LIN {X 0,Y 291.347,Z 435.191,A -85,B 0,C 180,E1 -16863.698,E2 -16863.698} C_VEL
LIN {X 0,Y 291.408,Z 435.188,A -85,B 0,C 180,E1 -16867.262,E2 -16867.262} C_VEL
LIN {X 0,Y 291.407,Z 435.186,A -85,B 0,C 180,E1 -16870.63,E2 -16870.63} C_VEL
LIN {X 0,Y 291.354,Z 435.191,A -85,B 0,C 180,E1 -16874.39,E2 -16874.39} C_VEL
LIN {X 0,Y 291.333,Z 435.194,A -85,B 0,C 180,E1 -16878.403,E2 -16878.403} C_VEL
LIN {X 0,Y 291.349,Z 435.194,A -85,B 0,C 180,E1 -16881.157,E2 -16881.157} C_VEL
LIN {X 0,Y 291.362,Z 435.192,A -85,B 0,C 180,E1 -16884.626,E2 -16884.626} C_VEL
LIN {X 0,Y 291.372,Z 435.186,A -85,B 0,C 180,E1 -16887.951,E2 -16887.951} C_VEL
LIN {X 0,Y 291.379,Z 435.188,A -85,B 0,C 180,E1 -16891.158,E2 -16891.158} C_VEL
LIN {X 0,Y 291.414,Z 435.184,A -85,B 0,C 180,E1 -16894.272,E2 -16894.272} C_VEL
LIN {X 0,Y 291.384,Z 435.184,A -85,B 0,C 180,E1 -16897.3,E2 -16897.3} C_VEL
LIN {X 0,Y 291.46,Z 435.179,A -85,B 0,C 180,E1 -16900.27,E2 -16900.27} C_VEL
LIN {X 0,Y 291.557,Z 435.169,A -85,B 0,C 180,E1 -16904.624,E2 -16904.624} C_VEL
LIN {X 0,Y 291.539,Z 435.169,A -85,B 0,C 180,E1 -16908.881,E2 -16908.881} C_VEL
LIN {X 0,Y 291.67,Z 435.151,A -85,B 0,C 180,E1 -16911.687,E2 -16911.687} C_VEL
LIN {X 0,Y 291.627,Z 435.154,A -85,B 0,C 180,E1 -16914.468,E2 -16914.468} C_VEL
LIN {X 0,Y 291.892,Z 435.126,A -85,B 0,C 180,E1 -16918.62,E2 -16918.62} C_VEL
LIN {X 0,Y 291.893,Z 435.118,A -85,B 0,C 180,E1 -16921.38,E2 -16921.38} C_VEL
LIN {X 0,Y 291.556,Z 435.166,A -85,B 0,C 180,E1 -16924.218,E2 -16924.218} C_VEL
LIN {X 0,Y 290.899,Z 435.248,A -85,B 0,C 180,E1 -16925.372,E2 -16925.372} C_VEL
LIN {X 0,Y 288.07,Z 435.598,A -85,B 0,C 180,E1 -16927.252,E2 -16927.252} C_VEL
LIN {X 0,Y 285.651,Z 435.902,A -85,B 0,C 180,E1 -16928.777,E2 -16928.777} C_VEL
LIN {X 0,Y 284.591,Z 436.034,A -85,B 0,C 180,E1 -16929.959,E2 -16929.959} C_VEL
LIN {X 0,Y 284.493,Z 436.044,A -85,B 0,C 180,E1 -16930.36,E2 -16930.36} C_VEL
LIN {X 0,Y 284.484,Z 436.05,A -85,B 0,C 180,E1 -16934.303,E2 -16934.303} C_VEL
LIN {X 0,Y 284.427,Z 436.051,A -85,B 0,C 180,E1 -16937.248,E2 -16937.248} C_VEL
LIN {X 0,Y 284.379,Z 436.064,A -85,B 0,C 180,E1 -16940.242,E2 -16940.242} C_VEL
LIN {X 0,Y 284.34,Z 436.065,A -85,B 0,C 180,E1 -16944.846,E2 -16944.846} C_VEL
LIN {X 0,Y 284.331,Z 436.069,A -85,B 0,C 180,E1 -16948.011,E2 -16948.011} C_VEL
LIN {X 0,Y 284.295,Z 436.072,A -85,B 0,C 180,E1 -16951.274,E2 -16951.274} C_VEL
LIN {X 0,Y 284.363,Z 436.065,A -85,B 0,C 180,E1 -16955.354,E2 -16955.354} C_VEL
LIN {X 0,Y 284.368,Z 436.211,A -85,B 0,C 180,E1 -16958.839,E2 -16958.839} C_VEL
LIN {X 0,Y 285.634,Z 442.53,A -85,B 0,C 180,E1 -16962.426,E2 -16962.426} C_VEL
LIN {X 0,Y 287.31,Z 450.763,A -85,B 0,C 180,E1 -16966.771,E2 -16966.771} C_VEL
LIN {X 0,Y 288.547,Z 457.203,A -85,B 0,C 180,E1 -16969.939,E2 -16969.939} C_VEL
LIN {X 0,Y 288.86,Z 459.714,A -85,B 0,C 180,E1 -16971.13,E2 -16971.13} C_VEL
LIN {X 0,Y 288.1,Z 465.339,A -85,B 0,C 180,E1 -16973.612,E2 -16973.612} C_VEL
LIN {X 0,Y 286.625,Z 474.02,A -85,B 0,C 180,E1 -16977.355,E2 -16977.355} C_VEL
LIN {X 0,Y 285.082,Z 485.04,A -85,B 0,C 180,E1 -16982.07,E2 -16982.07} C_VEL
LIN {X 0,Y 284.576,Z 489.714,A -85,B 0,C 180,E1 -16984.074,E2 -16984.074} C_VEL
LIN {X 0,Y 287.073,Z 505.085,A -85,B 0,C 180,E1 -16984.981,E2 -16984.981} C_VEL
LIN {X 0,Y 288.406,Z 518.048,A -85,B 0,C 180,E1 -16985.981,E2 -16985.981} C_VEL
LIN {X 0,Y 288.965,Z 530.807,A -85,B 0,C 180,E1 -16987.206,E2 -16987.206} C_VEL
LIN {X 0,Y 288.929,Z 542.594,A -85,B 0,C 180,E1 -16988.601,E2 -16988.601} C_VEL
LIN {X 0,Y 288.46,Z 553.824,A -85,B 0,C 180,E1 -16990.242,E2 -16990.242} C_VEL
LIN {X 0,Y 287.04,Z 562.869,A -85,B 0,C 180,E1 -16991.81,E2 -16991.81} C_VEL
LIN {X 0,Y 285.561,Z 571.816,A -85,B 0,C 180,E1 -16993.707,E2 -16993.707} C_VEL
LIN {X 0,Y 284.788,Z 576.889,A -85,B 0,C 180,E1 -16994.982,E2 -16994.982} C_VEL
LIN {X 0,Y 283.886,Z 583.999,A -85,B 0,C 180,E1 -16997.126,E2 -16997.126} C_VEL
LIN {X 0,Y 283.299,Z 589.729,A -85,B 0,C 180,E1 -16999.277,E2 -16999.277} C_VEL
LIN {X 0,Y 283.176,Z 594.281,A -85,B 0,C 180,E1 -17001.436,E2 -17001.436} C_VEL
LIN {X 0,Y 283.275,Z 596.802,A -85,B 0,C 180,E1 -17002.93,E2 -17002.93} C_VEL
LIN {X 0,Y 283.396,Z 598.695,A -85,B 0,C 180,E1 -17004.307,E2 -17004.307} C_VEL
LIN {X 0,Y 283.685,Z 600.209,A -85,B 0,C 180,E1 -17005.738,E2 -17005.738} C_VEL
LIN {X 0,Y 283.839,Z 601.281,A -85,B 0,C 180,E1 -17007.162,E2 -17007.162} C_VEL
LIN {X 0,Y 284.353,Z 602.219,A -85,B 0,C 180,E1 -17010,E2 -17010} C_VEL
LIN {X 0,Y 283.84,Z 601.271,A -85,B 0,C 180,E1 -17012.839,E2 -17012.839} C_VEL
LIN {X 0,Y 283.684,Z 600.194,A -85,B 0,C 180,E1 -17014.262,E2 -17014.262} C_VEL
LIN {X 0,Y 283.39,Z 598.672,A -85,B 0,C 180,E1 -17015.693,E2 -17015.693} C_VEL
LIN {X 0,Y 283.199,Z 595.541,A -85,B 0,C 180,E1 -17017.845,E2 -17017.845} C_VEL
LIN {X 0,Y 283.227,Z 591.348,A -85,B 0,C 180,E1 -17020.003,E2 -17020.003} C_VEL
LIN {X 0,Y 283.741,Z 584.975,A -85,B 0,C 180,E1 -17022.517,E2 -17022.517} C_VEL
LIN {X 0,Y 284.62,Z 578.08,A -85,B 0,C 180,E1 -17024.661,E2 -17024.661} C_VEL
LIN {X 0,Y 285.383,Z 572.557,A -85,B 0,C 180,E1 -17026.099,E2 -17026.099} C_VEL
LIN {X 0,Y 286.766,Z 564.569,A -85,B 0,C 180,E1 -17027.839,E2 -17027.839} C_VEL
LIN {X 0,Y 288.329,Z 554.77,A -85,B 0,C 180,E1 -17029.582,E2 -17029.582} C_VEL
LIN {X 0,Y 288.853,Z 543.762,A -85,B 0,C 180,E1 -17031.218,E2 -17031.218} C_VEL
LIN {X 0,Y 289.008,Z 533.538,A -85,B 0,C 180,E1 -17032.471,E2 -17032.471} C_VEL
LIN {X 0,Y 288.596,Z 521.211,A -85,B 0,C 180,E1 -17033.716,E2 -17033.716} C_VEL
LIN {X 0,Y 287.262,Z 507.25,A -85,B 0,C 180,E1 -17034.842,E2 -17034.842} C_VEL
LIN {X 0,Y 285.279,Z 494.142,A -85,B 0,C 180,E1 -17035.667,E2 -17035.667} C_VEL
LIN {X 0,Y 284.558,Z 489.7,A -85,B 0,C 180,E1 -17035.902,E2 -17035.902} C_VEL
LIN {X 0,Y 286.053,Z 477.671,A -85,B 0,C 180,E1 -17041.061,E2 -17041.061} C_VEL
LIN {X 0,Y 287.257,Z 470.208,A -85,B 0,C 180,E1 -17044.244,E2 -17044.244} C_VEL
LIN {X 0,Y 288.78,Z 461.165,A -85,B 0,C 180,E1 -17048.176,E2 -17048.176} C_VEL
LIN {X 0,Y 288.817,Z 458.788,A -85,B 0,C 180,E1 -17049.248,E2 -17049.248} C_VEL
LIN {X 0,Y 287.42,Z 451.508,A -85,B 0,C 180,E1 -17052.814,E2 -17052.814} C_VEL
LIN {X 0,Y 285.966,Z 444.403,A -85,B 0,C 180,E1 -17056.517,E2 -17056.517} C_VEL
LIN {X 0,Y 284.724,Z 437.997,A -85,B 0,C 180,E1 -17060.076,E2 -17060.076} C_VEL
LIN {X 0,Y 284.329,Z 436.071,A -85,B 0,C 180,E1 -17061.269,E2 -17061.269} C_VEL
LIN {X 0,Y 284.364,Z 436.063,A -85,B 0,C 180,E1 -17064.646,E2 -17064.646} C_VEL
LIN {X 0,Y 284.297,Z 436.069,A -85,B 0,C 180,E1 -17068.726,E2 -17068.726} C_VEL
LIN {X 0,Y 284.399,Z 436.06,A -85,B 0,C 180,E1 -17072.827,E2 -17072.827} C_VEL
LIN {X 0,Y 284.336,Z 436.065,A -85,B 0,C 180,E1 -17076.704,E2 -17076.704} C_VEL
LIN {X 0,Y 284.406,Z 436.057,A -85,B 0,C 180,E1 -17081.262,E2 -17081.262} C_VEL
LIN {X 0,Y 284.495,Z 436.047,A -85,B 0,C 180,E1 -17084.459,E2 -17084.459} C_VEL
LIN {X 0,Y 284.492,Z 436.047,A -85,B 0,C 180,E1 -17088.602,E2 -17088.602} C_VEL
LIN {X 0,Y 284.625,Z 436.032,A -85,B 0,C 180,E1 -17091.48,E2 -17091.48} C_VEL
LIN {X 0,Y 284.598,Z 436.034,A -85,B 0,C 180,E1 -17094.331,E2 -17094.331} C_VEL
LIN {X 0,Y 284.86,Z 436,A -85,B 0,C 180,E1 -17098.586,E2 -17098.586} C_VEL
LIN {X 0,Y 284.859,Z 436.002,A -85,B 0,C 180,E1 -17101.414,E2 -17101.414} C_VEL
LIN {X 0,Y 284.677,Z 436.023,A -85,B 0,C 180,E1 -17107.091,E2 -17107.091} C_VEL
LIN {X 0,Y 284.521,Z 436.042,A -85,B 0,C 180,E1 -17109.957,E2 -17109.957} C_VEL
LIN {X 0,Y 284.486,Z 436.028,A -85,B 0,C 180,E1 -17114.303,E2 -17114.303} C_VEL
LIN {X 0,Y 284.428,Z 436.036,A -85,B 0,C 180,E1 -17117.248,E2 -17117.248} C_VEL
LIN {X 0,Y 284.382,Z 436.056,A -85,B 0,C 180,E1 -17120.242,E2 -17120.242} C_VEL
LIN {X 0,Y 284.372,Z 436.056,A -85,B 0,C 180,E1 -17123.875,E2 -17123.875} C_VEL
LIN {X 0,Y 284.397,Z 436.041,A -85,B 0,C 180,E1 -17127.172,E2 -17127.172} C_VEL
LIN {X 0,Y 284.296,Z 436.069,A -85,B 0,C 180,E1 -17131.274,E2 -17131.274} C_VEL
LIN {X 0,Y 284.343,Z 436.064,A -85,B 0,C 180,E1 -17135.348,E2 -17135.348} C_VEL
LIN {X 0,Y 284.311,Z 436.068,A -85,B 0,C 180,E1 -17138.169,E2 -17138.169} C_VEL
LIN {X 0,Y 284.286,Z 436.071,A -85,B 0,C 180,E1 -17142.128,E2 -17142.128} C_VEL
LIN {X 0,Y 284.32,Z 436.066,A -85,B 0,C 180,E1 -17146.201,E2 -17146.201} C_VEL
LIN {X 0,Y 284.354,Z 436.06,A -85,B 0,C 180,E1 -17150.013,E2 -17150.013} C_VEL
LIN {X 0,Y 284.358,Z 436.059,A -85,B 0,C 180,E1 -17153.618,E2 -17153.618} C_VEL
LIN {X 0,Y 284.31,Z 436.069,A -85,B 0,C 180,E1 -17157.19,E2 -17157.19} C_VEL
LIN {X 0,Y 284.358,Z 436.063,A -85,B 0,C 180,E1 -17160.376,E2 -17160.376} C_VEL
LIN {X 0,Y 284.389,Z 436.062,A -85,B 0,C 180,E1 -17164.375,E2 -17164.375} C_VEL
LIN {X 0,Y 284.416,Z 436.147,A -85,B 0,C 180,E1 -17165.136,E2 -17165.136} C_VEL
LIN {X 0,Y 287.692,Z 444.694,A -85,B 0,C 180,E1 -17166.157,E2 -17166.157} C_VEL
LIN {X 0,Y 291.581,Z 455.705,A -85,B 0,C 180,E1 -17167.66,E2 -17167.66} C_VEL
LIN {X 0,Y 294.434,Z 465.794,A -85,B 0,C 180,E1 -17169.236,E2 -17169.236} C_VEL
LIN {X 0,Y 294.248,Z 468.913,A -85,B 0,C 180,E1 -17169.676,E2 -17169.676} C_VEL
LIN {X 0,Y 292.847,Z 478.165,A -85,B 0,C 180,E1 -17171.096,E2 -17171.096} C_VEL
LIN {X 0,Y 291.409,Z 487.197,A -85,B 0,C 180,E1 -17172.816,E2 -17172.816} C_VEL
LIN {X 0,Y 289.663,Z 495.979,A -85,B 0,C 180,E1 -17174.881,E2 -17174.881} C_VEL
LIN {X 0,Y 288.283,Z 503.021,A -85,B 0,C 180,E1 -17176.967,E2 -17176.967} C_VEL
LIN {X 0,Y 287.359,Z 507.755,A -85,B 0,C 180,E1 -17178.717,E2 -17178.717} C_VEL
LIN {X 0,Y 286.426,Z 512.352,A -85,B 0,C 180,E1 -17180.823,E2 -17180.823} C_VEL
LIN {X 0,Y 285.582,Z 515.883,A -85,B 0,C 180,E1 -17182.932,E2 -17182.932} C_VEL
LIN {X 0,Y 285.161,Z 517.704,A -85,B 0,C 180,E1 -17184.342,E2 -17184.342} C_VEL
LIN {X 0,Y 284.821,Z 519.076,A -85,B 0,C 180,E1 -17185.755,E2 -17185.755} C_VEL
LIN {X 0,Y 284.762,Z 520.603,A -85,B 0,C 180,E1 -17188.586,E2 -17188.586} C_VEL
LIN {X 0,Y 284.742,Z 520.826,A -85,B 0,C 180,E1 -17190,E2 -17190} C_VEL
LIN {X 0,Y 284.761,Z 520.64,A -85,B 0,C 180,E1 -17191.414,E2 -17191.414} C_VEL
LIN {X 0,Y 284.812,Z 519.162,A -85,B 0,C 180,E1 -17194.245,E2 -17194.245} C_VEL
LIN {X 0,Y 285.147,Z 517.83,A -85,B 0,C 180,E1 -17195.658,E2 -17195.658} C_VEL
LIN {X 0,Y 285.867,Z 515.009,A -85,B 0,C 180,E1 -17197.771,E2 -17197.771} C_VEL
LIN {X 0,Y 286.759,Z 511.19,A -85,B 0,C 180,E1 -17199.878,E2 -17199.878} C_VEL
LIN {X 0,Y 287.795,Z 505.275,A -85,B 0,C 180,E1 -17202.363,E2 -17202.363} C_VEL
LIN {X 0,Y 289.175,Z 498.879,A -85,B 0,C 180,E1 -17204.425,E2 -17204.425} C_VEL
LIN {X 0,Y 290.779,Z 490.841,A -85,B 0,C 180,E1 -17206.499,E2 -17206.499} C_VEL
LIN {X 0,Y 292.119,Z 482.62,A -85,B 0,C 180,E1 -17208.226,E2 -17208.226} C_VEL
LIN {X 0,Y 293.692,Z 472.862,A -85,B 0,C 180,E1 -17209.867,E2 -17209.867} C_VEL
LIN {X 0,Y 294.51,Z 466.371,A -85,B 0,C 180,E1 -17210.791,E2 -17210.791} C_VEL
LIN {X 0,Y 291.709,Z 456.12,A -85,B 0,C 180,E1 -17212.399,E2 -17212.399} C_VEL
LIN {X 0,Y 288.801,Z 447.537,A -85,B 0,C 180,E1 -17213.592,E2 -17213.592} C_VEL
LIN {X 0,Y 284.726,Z 437.456,A -85,B 0,C 180,E1 -17214.859,E2 -17214.859} C_VEL
LIN {X 0,Y 284.419,Z 436.058,A -85,B 0,C 180,E1 -17215.034,E2 -17215.034} C_VEL
LIN {X 0,Y 284.33,Z 436.06,A -85,B 0,C 180,E1 -17218.011,E2 -17218.011} C_VEL
LIN {X 0,Y 284.296,Z 436.07,A -85,B 0,C 180,E1 -17221.274,E2 -17221.274} C_VEL
LIN {X 0,Y 284.364,Z 436.063,A -85,B 0,C 180,E1 -17225.354,E2 -17225.354} C_VEL
LIN {X 0,Y 284.341,Z 436.065,A -85,B 0,C 180,E1 -17228.165,E2 -17228.165} C_VEL
LIN {X 0,Y 284.344,Z 436.064,A -85,B 0,C 180,E1 -17232.141,E2 -17232.141} C_VEL
LIN {X 0,Y 284.298,Z 436.07,A -85,B 0,C 180,E1 -17236.197,E2 -17236.197} C_VEL
LIN {X 0,Y 284.308,Z 436.068,A -85,B 0,C 180,E1 -17240.024,E2 -17240.024} C_VEL
LIN {X 0,Y 284.332,Z 436.065,A -85,B 0,C 180,E1 -17243.614,E2 -17243.614} C_VEL
LIN {X 0,Y 284.309,Z 436.067,A -85,B 0,C 180,E1 -17247.19,E2 -17247.19} C_VEL
LIN {X 0,Y 284.357,Z 436.064,A -85,B 0,C 180,E1 -17250.376,E2 -17250.376} C_VEL
LIN {X 0,Y 284.376,Z 436.059,A -85,B 0,C 180,E1 -17253.586,E2 -17253.586} C_VEL
LIN {X 0,Y 284.368,Z 436.062,A -85,B 0,C 180,E1 -17256.707,E2 -17256.707} C_VEL
LIN {X 0,Y 284.406,Z 436.055,A -85,B 0,C 180,E1 -17261.262,E2 -17261.262} C_VEL
LIN {X 0,Y 284.494,Z 436.047,A -85,B 0,C 180,E1 -17264.459,E2 -17264.459} C_VEL
LIN {X 0,Y 284.491,Z 436.046,A -85,B 0,C 180,E1 -17268.601,E2 -17268.601} C_VEL
LIN {X 0,Y 284.624,Z 436.029,A -85,B 0,C 180,E1 -17271.48,E2 -17271.48} C_VEL
LIN {X 0,Y 284.597,Z 436.029,A -85,B 0,C 180,E1 -17274.331,E2 -17274.331} C_VEL
LIN {X 0,Y 284.858,Z 436.003,A -85,B 0,C 180,E1 -17278.586,E2 -17278.586} C_VEL
LIN {X 0,Y 284.859,Z 435.994,A -85,B 0,C 180,E1 -17281.414,E2 -17281.414} C_VEL
LIN {X 0,Y 284.676,Z 436.019,A -85,B 0,C 180,E1 -17287.091,E2 -17287.091} C_VEL
LIN {X 0,Y 284.493,Z 436.044,A -85,B 0,C 180,E1 -17290.36,E2 -17290.36} C_VEL
LIN {X 0,Y 283.799,Z 436.132,A -85,B 0,C 180,E1 -17291.541,E2 -17291.541} C_VEL
LIN {X 0,Y 280.951,Z 436.486,A -85,B 0,C 180,E1 -17293.466,E2 -17293.466} C_VEL
LIN {X 0,Y 278.535,Z 436.789,A -85,B 0,C 180,E1 -17295.029,E2 -17295.029} C_VEL
LIN {X 0,Y 277.474,Z 436.921,A -85,B 0,C 180,E1 -17296.239,E2 -17296.239} C_VEL
LIN {X 0,Y 277.373,Z 436.93,A -85,B 0,C 180,E1 -17296.65,E2 -17296.65} C_VEL
LIN {X 0,Y 277.292,Z 436.944,A -85,B 0,C 180,E1 -17300.783,E2 -17300.783} C_VEL
LIN {X 0,Y 277.294,Z 436.947,A -85,B 0,C 180,E1 -17304.158,E2 -17304.158} C_VEL
LIN {X 0,Y 277.326,Z 436.94,A -85,B 0,C 180,E1 -17307.505,E2 -17307.505} C_VEL
LIN {X 0,Y 277.273,Z 436.948,A -85,B 0,C 180,E1 -17310.481,E2 -17310.481} C_VEL
LIN {X 0,Y 277.255,Z 436.95,A -85,B 0,C 180,E1 -17313.895,E2 -17313.895} C_VEL
LIN {X 0,Y 277.283,Z 436.946,A -85,B 0,C 180,E1 -17317.467,E2 -17317.467} C_VEL
LIN {X 0,Y 277.322,Z 437.139,A -85,B 0,C 180,E1 -17318.222,E2 -17318.222} C_VEL
LIN {X 0,Y 278.6,Z 443.48,A -85,B 0,C 180,E1 -17321.951,E2 -17321.951} C_VEL
LIN {X 0,Y 280.048,Z 450.645,A -85,B 0,C 180,E1 -17325.874,E2 -17325.874} C_VEL
LIN {X 0,Y 281.663,Z 459.053,A -85,B 0,C 180,E1 -17330.156,E2 -17330.156} C_VEL
LIN {X 0,Y 281.813,Z 461.726,A -85,B 0,C 180,E1 -17331.43,E2 -17331.43} C_VEL
LIN {X 0,Y 280.511,Z 469.265,A -85,B 0,C 180,E1 -17334.813,E2 -17334.813} C_VEL
LIN {X 0,Y 278.965,Z 478.58,A -85,B 0,C 180,E1 -17338.933,E2 -17338.933} C_VEL
LIN {X 0,Y 277.645,Z 488.643,A -85,B 0,C 180,E1 -17343.379,E2 -17343.379} C_VEL
LIN {X 0,Y 280.156,Z 503.724,A -85,B 0,C 180,E1 -17344.303,E2 -17344.303} C_VEL
LIN {X 0,Y 281.504,Z 516.559,A -85,B 0,C 180,E1 -17345.318,E2 -17345.318} C_VEL
LIN {X 0,Y 282.114,Z 528.716,A -85,B 0,C 180,E1 -17346.51,E2 -17346.51} C_VEL
LIN {X 0,Y 282.129,Z 540.026,A -85,B 0,C 180,E1 -17347.859,E2 -17347.859} C_VEL
LIN {X 0,Y 281.677,Z 550.499,A -85,B 0,C 180,E1 -17349.364,E2 -17349.364} C_VEL
LIN {X 0,Y 281.112,Z 557.048,A -85,B 0,C 180,E1 -17350.465,E2 -17350.465} C_VEL
LIN {X 0,Y 279.385,Z 567.046,A -85,B 0,C 180,E1 -17352.43,E2 -17352.43} C_VEL
LIN {X 0,Y 277.789,Z 575.855,A -85,B 0,C 180,E1 -17354.595,E2 -17354.595} C_VEL
LIN {X 0,Y 276.862,Z 582.969,A -85,B 0,C 180,E1 -17356.794,E2 -17356.794} C_VEL
LIN {X 0,Y 276.249,Z 588.704,A -85,B 0,C 180,E1 -17359,E2 -17359} C_VEL
LIN {X 0,Y 276.115,Z 593.26,A -85,B 0,C 180,E1 -17361.216,E2 -17361.216} C_VEL
LIN {X 0,Y 276.204,Z 596.035,A -85,B 0,C 180,E1 -17362.912,E2 -17362.912} C_VEL
LIN {X 0,Y 276.599,Z 599.193,A -85,B 0,C 180,E1 -17365.628,E2 -17365.628} C_VEL
LIN {X 0,Y 276.783,Z 600.271,A -85,B 0,C 180,E1 -17367.089,E2 -17367.089} C_VEL
LIN {X 0,Y 277.321,Z 601.213,A -85,B 0,C 180,E1 -17370,E2 -17370} C_VEL
LIN {X 0,Y 276.783,Z 600.26,A -85,B 0,C 180,E1 -17372.911,E2 -17372.911} C_VEL
LIN {X 0,Y 276.597,Z 599.177,A -85,B 0,C 180,E1 -17374.372,E2 -17374.372} C_VEL
LIN {X 0,Y 276.208,Z 595.994,A -85,B 0,C 180,E1 -17377.095,E2 -17377.095} C_VEL
LIN {X 0,Y 276.121,Z 591.827,A -85,B 0,C 180,E1 -17379.523,E2 -17379.523} C_VEL
LIN {X 0,Y 276.403,Z 586.875,A -85,B 0,C 180,E1 -17381.737,E2 -17381.737} C_VEL
LIN {X 0,Y 277.27,Z 579.519,A -85,B 0,C 180,E1 -17384.308,E2 -17384.308} C_VEL
LIN {X 0,Y 278.203,Z 573.005,A -85,B 0,C 180,E1 -17386.134,E2 -17386.134} C_VEL
LIN {X 0,Y 279.649,Z 565.264,A -85,B 0,C 180,E1 -17387.931,E2 -17387.931} C_VEL
LIN {X 0,Y 281.203,Z 555.896,A -85,B 0,C 180,E1 -17389.719,E2 -17389.719} C_VEL
LIN {X 0,Y 281.922,Z 545.374,A -85,B 0,C 180,E1 -17391.382,E2 -17391.382} C_VEL
LIN {X 0,Y 282.183,Z 534.115,A -85,B 0,C 180,E1 -17392.851,E2 -17392.851} C_VEL
LIN {X 0,Y 281.879,Z 522.439,A -85,B 0,C 180,E1 -17394.107,E2 -17394.107} C_VEL
LIN {X 0,Y 280.911,Z 510.397,A -85,B 0,C 180,E1 -17395.171,E2 -17395.171} C_VEL
LIN {X 0,Y 279.154,Z 497.2,A -85,B 0,C 180,E1 -17396.097,E2 -17396.097} C_VEL
LIN {X 0,Y 277.639,Z 488.645,A -85,B 0,C 180,E1 -17396.583,E2 -17396.583} C_VEL
LIN {X 0,Y 278.951,Z 478.521,A -85,B 0,C 180,E1 -17401.062,E2 -17401.062} C_VEL
LIN {X 0,Y 280.494,Z 469.171,A -85,B 0,C 180,E1 -17405.19,E2 -17405.19} C_VEL
LIN {X 0,Y 281.814,Z 461.628,A -85,B 0,C 180,E1 -17408.57,E2 -17408.57} C_VEL
LIN {X 0,Y 281.66,Z 458.923,A -85,B 0,C 180,E1 -17409.844,E2 -17409.844} C_VEL
LIN {X 0,Y 280.328,Z 452.037,A -85,B 0,C 180,E1 -17413.36,E2 -17413.36} C_VEL
LIN {X 0,Y 278.862,Z 445.062,A -85,B 0,C 180,E1 -17417.12,E2 -17417.12} C_VEL
LIN {X 0,Y 277.662,Z 438.766,A -85,B 0,C 180,E1 -17420.744,E2 -17420.744} C_VEL
LIN {X 0,Y 277.291,Z 436.949,A -85,B 0,C 180,E1 -17421.91,E2 -17421.91} C_VEL
LIN {X 0,Y 277.306,Z 436.943,A -85,B 0,C 180,E1 -17424.345,E2 -17424.345} C_VEL
LIN {X 0,Y 277.246,Z 436.952,A -85,B 0,C 180,E1 -17427.837,E2 -17427.837} C_VEL
LIN {X 0,Y 277.271,Z 436.948,A -85,B 0,C 180,E1 -17431.21,E2 -17431.21} C_VEL
LIN {X 0,Y 277.312,Z 436.94,A -85,B 0,C 180,E1 -17434.479,E2 -17434.479} C_VEL
LIN {X 0,Y 277.271,Z 436.946,A -85,B 0,C 180,E1 -17437.654,E2 -17437.654} C_VEL
LIN {X 0,Y 277.347,Z 436.935,A -85,B 0,C 180,E1 -17440.766,E2 -17440.766} C_VEL
LIN {X 0,Y 277.438,Z 436.927,A -85,B 0,C 180,E1 -17445.326,E2 -17445.326} C_VEL
LIN {X 0,Y 277.463,Z 436.927,A -85,B 0,C 180,E1 -17449.787,E2 -17449.787} C_VEL
LIN {X 0,Y 277.632,Z 436.902,A -85,B 0,C 180,E1 -17452.729,E2 -17452.729} C_VEL
LIN {X 0,Y 277.826,Z 436.877,A -85,B 0,C 180,E1 -17458.551,E2 -17458.551} C_VEL
LIN {X 0,Y 277.825,Z 436.879,A -85,B 0,C 180,E1 -17461.45,E2 -17461.45} C_VEL
LIN {X 0,Y 277.631,Z 436.902,A -85,B 0,C 180,E1 -17467.272,E2 -17467.272} C_VEL
LIN {X 0,Y 277.464,Z 436.92,A -85,B 0,C 180,E1 -17470.213,E2 -17470.213} C_VEL
LIN {X 0,Y 277.438,Z 436.904,A -85,B 0,C 180,E1 -17474.674,E2 -17474.674} C_VEL
LIN {X 0,Y 277.348,Z 436.928,A -85,B 0,C 180,E1 -17479.234,E2 -17479.234} C_VEL
LIN {X 0,Y 277.322,Z 436.933,A -85,B 0,C 180,E1 -17484.17,E2 -17484.17} C_VEL
LIN {X 0,Y 277.325,Z 436.918,A -85,B 0,C 180,E1 -17487.504,E2 -17487.504} C_VEL
LIN {X 0,Y 277.274,Z 436.937,A -85,B 0,C 180,E1 -17490.481,E2 -17490.481} C_VEL
LIN {X 0,Y 277.249,Z 436.946,A -85,B 0,C 180,E1 -17493.896,E2 -17493.896} C_VEL
LIN {X 0,Y 277.268,Z 436.948,A -85,B 0,C 180,E1 -17497.47,E2 -17497.47} C_VEL
LIN {X 0,Y 277.218,Z 436.955,A -85,B 0,C 180,E1 -17501.235,E2 -17501.235} C_VEL
LIN {X 0,Y 277.249,Z 436.951,A -85,B 0,C 180,E1 -17505.217,E2 -17505.217} C_VEL
LIN {X 0,Y 277.297,Z 436.94,A -85,B 0,C 180,E1 -17509.494,E2 -17509.494} C_VEL
LIN {X 0,Y 277.294,Z 436.941,A -85,B 0,C 180,E1 -17512.535,E2 -17512.535} C_VEL
LIN {X 0,Y 277.257,Z 436.943,A -85,B 0,C 180,E1 -17516.105,E2 -17516.105} C_VEL
LIN {X 0,Y 277.264,Z 436.946,A -85,B 0,C 180,E1 -17519.539,E2 -17519.539} C_VEL
LIN {X 0,Y 277.346,Z 436.939,A -85,B 0,C 180,E1 -17523.675,E2 -17523.675} C_VEL
LIN {X 0,Y 277.356,Z 436.937,A -85,B 0,C 180,E1 -17524.433,E2 -17524.433} C_VEL
LIN {X 0,Y 281.583,Z 447.834,A -85,B 0,C 180,E1 -17525.806,E2 -17525.806} C_VEL
LIN {X 0,Y 285.395,Z 458.984,A -85,B 0,C 180,E1 -17527.436,E2 -17527.436} C_VEL
LIN {X 0,Y 287.67,Z 467.111,A -85,B 0,C 180,E1 -17528.766,E2 -17528.766} C_VEL
LIN {X 0,Y 287.86,Z 468.825,A -85,B 0,C 180,E1 -17529.044,E2 -17529.044} C_VEL
LIN {X 0,Y 286.208,Z 479.174,A -85,B 0,C 180,E1 -17530.64,E2 -17530.64} C_VEL
LIN {X 0,Y 284.703,Z 488.204,A -85,B 0,C 180,E1 -17532.398,E2 -17532.398} C_VEL
LIN {X 0,Y 282.885,Z 496.986,A -85,B 0,C 180,E1 -17534.51,E2 -17534.51} C_VEL
LIN {X 0,Y 281.441,Z 504.028,A -85,B 0,C 180,E1 -17536.645,E2 -17536.645} C_VEL
LIN {X 0,Y 280.47,Z 508.762,A -85,B 0,C 180,E1 -17538.436,E2 -17538.436} C_VEL
LIN {X 0,Y 279.491,Z 513.358,A -85,B 0,C 180,E1 -17540.593,E2 -17540.593} C_VEL
LIN {X 0,Y 278.609,Z 516.889,A -85,B 0,C 180,E1 -17542.754,E2 -17542.754} C_VEL
LIN {X 0,Y 278.168,Z 518.71,A -85,B 0,C 180,E1 -17544.2,E2 -17544.2} C_VEL
LIN {X 0,Y 277.813,Z 520.081,A -85,B 0,C 180,E1 -17545.647,E2 -17545.647} C_VEL
LIN {X 0,Y 277.739,Z 521.608,A -85,B 0,C 180,E1 -17548.55,E2 -17548.55} C_VEL
LIN {X 0,Y 277.717,Z 521.83,A -85,B 0,C 180,E1 -17550,E2 -17550} C_VEL
LIN {X 0,Y 277.738,Z 521.645,A -85,B 0,C 180,E1 -17551.45,E2 -17551.45} C_VEL
LIN {X 0,Y 277.804,Z 520.167,A -85,B 0,C 180,E1 -17554.353,E2 -17554.353} C_VEL
LIN {X 0,Y 278.153,Z 518.834,A -85,B 0,C 180,E1 -17555.8,E2 -17555.8} C_VEL
LIN {X 0,Y 278.906,Z 516.013,A -85,B 0,C 180,E1 -17557.966,E2 -17557.966} C_VEL
LIN {X 0,Y 279.838,Z 512.193,A -85,B 0,C 180,E1 -17560.125,E2 -17560.125} C_VEL
LIN {X 0,Y 280.933,Z 506.282,A -85,B 0,C 180,E1 -17562.668,E2 -17562.668} C_VEL
LIN {X 0,Y 282.374,Z 499.882,A -85,B 0,C 180,E1 -17564.78,E2 -17564.78} C_VEL
LIN {X 0,Y 284.048,Z 491.844,A -85,B 0,C 180,E1 -17566.901,E2 -17566.901} C_VEL
LIN {X 0,Y 285.452,Z 483.622,A -85,B 0,C 180,E1 -17568.667,E2 -17568.667} C_VEL
LIN {X 0,Y 287.075,Z 473.992,A -85,B 0,C 180,E1 -17570.324,E2 -17570.324} C_VEL
LIN {X 0,Y 287.801,Z 467.702,A -85,B 0,C 180,E1 -17571.253,E2 -17571.253} C_VEL
LIN {X 0,Y 284.865,Z 457.151,A -85,B 0,C 180,E1 -17572.97,E2 -17572.97} C_VEL
LIN {X 0,Y 281.34,Z 447.265,A -85,B 0,C 180,E1 -17574.399,E2 -17574.399} C_VEL
LIN {X 0,Y 277.338,Z 436.938,A -85,B 0,C 180,E1 -17575.719,E2 -17575.719} C_VEL
LIN {X 0,Y 277.27,Z 436.936,A -85,B 0,C 180,E1 -17578.79,E2 -17578.79} C_VEL
LIN {X 0,Y 277.246,Z 436.944,A -85,B 0,C 180,E1 -17582.163,E2 -17582.163} C_VEL
LIN {X 0,Y 277.329,Z 436.938,A -85,B 0,C 180,E1 -17585.812,E2 -17585.812} C_VEL
LIN {X 0,Y 277.288,Z 436.946,A -85,B 0,C 180,E1 -17589.319,E2 -17589.319} C_VEL
LIN {X 0,Y 277.265,Z 436.949,A -85,B 0,C 180,E1 -17593.187,E2 -17593.187} C_VEL
LIN {X 0,Y 277.234,Z 436.951,A -85,B 0,C 180,E1 -17597.321,E2 -17597.321} C_VEL
LIN {X 0,Y 277.263,Z 436.946,A -85,B 0,C 180,E1 -17601.793,E2 -17601.793} C_VEL
LIN {X 0,Y 277.285,Z 436.943,A -85,B 0,C 180,E1 -17604.341,E2 -17604.341} C_VEL
LIN {X 0,Y 277.245,Z 436.945,A -85,B 0,C 180,E1 -17607.836,E2 -17607.836} C_VEL
LIN {X 0,Y 277.269,Z 436.945,A -85,B 0,C 180,E1 -17611.21,E2 -17611.21} C_VEL
LIN {X 0,Y 277.313,Z 436.941,A -85,B 0,C 180,E1 -17614.479,E2 -17614.479} C_VEL
LIN {X 0,Y 277.288,Z 436.939,A -85,B 0,C 180,E1 -17617.655,E2 -17617.655} C_VEL
LIN {X 0,Y 277.347,Z 436.938,A -85,B 0,C 180,E1 -17620.766,E2 -17620.766} C_VEL
LIN {X 0,Y 277.437,Z 436.924,A -85,B 0,C 180,E1 -17625.326,E2 -17625.326} C_VEL
LIN {X 0,Y 277.462,Z 436.92,A -85,B 0,C 180,E1 -17629.787,E2 -17629.787} C_VEL
LIN {X 0,Y 277.631,Z 436.899,A -85,B 0,C 180,E1 -17632.728,E2 -17632.728} C_VEL
LIN {X 0,Y 277.824,Z 436.879,A -85,B 0,C 180,E1 -17638.55,E2 -17638.55} C_VEL
LIN {X 0,Y 277.824,Z 436.87,A -85,B 0,C 180,E1 -17641.449,E2 -17641.449} C_VEL
LIN {X 0,Y 277.631,Z 436.896,A -85,B 0,C 180,E1 -17647.271,E2 -17647.271} C_VEL
LIN {X 0,Y 277.453,Z 436.924,A -85,B 0,C 180,E1 -17650.34,E2 -17650.34} C_VEL
LIN {X 0,Y 277.437,Z 436.926,A -85,B 0,C 180,E1 -17654.674,E2 -17654.674} C_VEL
LIN {X 0,Y 277.373,Z 436.93,A -85,B 0,C 180,E1 -17656.65,E2 -17656.65} C_VEL
LIN {X 0,Y 276.664,Z 437.022,A -85,B 0,C 180,E1 -17657.862,E2 -17657.862} C_VEL
LIN {X 0,Y 273.783,Z 437.382,A -85,B 0,C 180,E1 -17659.836,E2 -17659.836} C_VEL
LIN {X 0,Y 271.353,Z 437.687,A -85,B 0,C 180,E1 -17661.44,E2 -17661.44} C_VEL
LIN {X 0,Y 270.3,Z 437.816,A -85,B 0,C 180,E1 -17662.683,E2 -17662.683} C_VEL
LIN {X 0,Y 270.206,Z 437.825,A -85,B 0,C 180,E1 -17663.105,E2 -17663.105} C_VEL
LIN {X 0,Y 270.263,Z 437.822,A -85,B 0,C 180,E1 -17666.236,E2 -17666.236} C_VEL
LIN {X 0,Y 270.197,Z 437.827,A -85,B 0,C 180,E1 -17669.617,E2 -17669.617} C_VEL
LIN {X 0,Y 270.221,Z 437.827,A -85,B 0,C 180,E1 -17673.668,E2 -17673.668} C_VEL
LIN {X 0,Y 270.238,Z 437.835,A -85,B 0,C 180,E1 -17677.438,E2 -17677.438} C_VEL
LIN {X 0,Y 271.516,Z 444.254,A -85,B 0,C 180,E1 -17681.354,E2 -17681.354} C_VEL
LIN {X 0,Y 272.818,Z 450.809,A -85,B 0,C 180,E1 -17685.072,E2 -17685.072} C_VEL
LIN {X 0,Y 274.316,Z 458.364,A -85,B 0,C 180,E1 -17689.094,E2 -17689.094} C_VEL
LIN {X 0,Y 274.756,Z 460.638,A -85,B 0,C 180,E1 -17690.247,E2 -17690.247} C_VEL
LIN {X 0,Y 274.838,Z 462.61,A -85,B 0,C 180,E1 -17691.208,E2 -17691.208} C_VEL
LIN {X 0,Y 273.881,Z 468.232,A -85,B 0,C 180,E1 -17693.829,E2 -17693.829} C_VEL
LIN {X 0,Y 272.23,Z 477.198,A -85,B 0,C 180,E1 -17697.919,E2 -17697.919} C_VEL
LIN {X 0,Y 270.883,Z 486.504,A -85,B 0,C 180,E1 -17702.16,E2 -17702.16} C_VEL
LIN {X 0,Y 270.76,Z 487.588,A -85,B 0,C 180,E1 -17702.656,E2 -17702.656} C_VEL
LIN {X 0,Y 273.285,Z 502.453,A -85,B 0,C 180,E1 -17703.597,E2 -17703.597} C_VEL
LIN {X 0,Y 274.696,Z 515.492,A -85,B 0,C 180,E1 -17704.664,E2 -17704.664} C_VEL
LIN {X 0,Y 275.349,Z 527.665,A -85,B 0,C 180,E1 -17705.897,E2 -17705.897} C_VEL
LIN {X 0,Y 275.317,Z 538.841,A -85,B 0,C 180,E1 -17707.263,E2 -17707.263} C_VEL
LIN {X 0,Y 274.833,Z 549.454,A -85,B 0,C 180,E1 -17708.826,E2 -17708.826} C_VEL
LIN {X 0,Y 274.188,Z 557.019,A -85,B 0,C 180,E1 -17710.146,E2 -17710.146} C_VEL
LIN {X 0,Y 272.553,Z 566.022,A -85,B 0,C 180,E1 -17711.975,E2 -17711.975} C_VEL
LIN {X 0,Y 271.105,Z 573.205,A -85,B 0,C 180,E1 -17713.746,E2 -17713.746} C_VEL
LIN {X 0,Y 270.024,Z 580.883,A -85,B 0,C 180,E1 -17716.069,E2 -17716.069} C_VEL
LIN {X 0,Y 269.397,Z 585.915,A -85,B 0,C 180,E1 -17717.954,E2 -17717.954} C_VEL
LIN {X 0,Y 269.073,Z 590.854,A -85,B 0,C 180,E1 -17720.225,E2 -17720.225} C_VEL
LIN {X 0,Y 269.134,Z 595.247,A -85,B 0,C 180,E1 -17722.89,E2 -17722.89} C_VEL
LIN {X 0,Y 269.516,Z 598.177,A -85,B 0,C 180,E1 -17725.513,E2 -17725.513} C_VEL
LIN {X 0,Y 269.723,Z 599.26,A -85,B 0,C 180,E1 -17727.013,E2 -17727.013} C_VEL
LIN {X 0,Y 270.288,Z 600.207,A -85,B 0,C 180,E1 -17730,E2 -17730} C_VEL
LIN {X 0,Y 269.723,Z 599.248,A -85,B 0,C 180,E1 -17732.987,E2 -17732.987} C_VEL
LIN {X 0,Y 269.514,Z 598.161,A -85,B 0,C 180,E1 -17734.487,E2 -17734.487} C_VEL
LIN {X 0,Y 269.15,Z 595.183,A -85,B 0,C 180,E1 -17737.137,E2 -17737.137} C_VEL
LIN {X 0,Y 269.074,Z 590.803,A -85,B 0,C 180,E1 -17739.775,E2 -17739.775} C_VEL
LIN {X 0,Y 269.398,Z 585.849,A -85,B 0,C 180,E1 -17742.047,E2 -17742.047} C_VEL
LIN {X 0,Y 270.344,Z 578.495,A -85,B 0,C 180,E1 -17744.683,E2 -17744.683} C_VEL
LIN {X 0,Y 271.37,Z 571.985,A -85,B 0,C 180,E1 -17746.552,E2 -17746.552} C_VEL
LIN {X 0,Y 272.83,Z 564.235,A -85,B 0,C 180,E1 -17748.395,E2 -17748.395} C_VEL
LIN {X 0,Y 274.454,Z 554.866,A -85,B 0,C 180,E1 -17750.225,E2 -17750.225} C_VEL
LIN {X 0,Y 275.119,Z 544.323,A -85,B 0,C 180,E1 -17751.938,E2 -17751.938} C_VEL
LIN {X 0,Y 275.369,Z 532.415,A -85,B 0,C 180,E1 -17753.527,E2 -17753.527} C_VEL
LIN {X 0,Y 274.995,Z 520.325,A -85,B 0,C 180,E1 -17754.851,E2 -17754.851} C_VEL
LIN {X 0,Y 273.838,Z 507.207,A -85,B 0,C 180,E1 -17756.011,E2 -17756.011} C_VEL
LIN {X 0,Y 271.902,Z 493.881,A -85,B 0,C 180,E1 -17756.944,E2 -17756.944} C_VEL
LIN {X 0,Y 270.738,Z 487.508,A -85,B 0,C 180,E1 -17757.349,E2 -17757.349} C_VEL
LIN {X 0,Y 272.229,Z 477.127,A -85,B 0,C 180,E1 -17762.08,E2 -17762.08} C_VEL
LIN {X 0,Y 273.844,Z 468.108,A -85,B 0,C 180,E1 -17766.177,E2 -17766.177} C_VEL
LIN {X 0,Y 274.838,Z 462.497,A -85,B 0,C 180,E1 -17768.793,E2 -17768.793} C_VEL
LIN {X 0,Y 274.305,Z 458.264,A -85,B 0,C 180,E1 -17770.904,E2 -17770.904} C_VEL
LIN {X 0,Y 272.796,Z 450.72,A -85,B 0,C 180,E1 -17774.933,E2 -17774.933} C_VEL
LIN {X 0,Y 271.217,Z 442.52,A -85,B 0,C 180,E1 -17779.622,E2 -17779.622} C_VEL
LIN {X 0,Y 270.237,Z 437.826,A -85,B 0,C 180,E1 -17782.561,E2 -17782.561} C_VEL
LIN {X 0,Y 270.206,Z 437.826,A -85,B 0,C 180,E1 -17786.893,E2 -17786.893} C_VEL
LIN {X 0,Y 270.198,Z 437.831,A -85,B 0,C 180,E1 -17790.383,E2 -17790.383} C_VEL
LIN {X 0,Y 270.264,Z 437.822,A -85,B 0,C 180,E1 -17793.764,E2 -17793.764} C_VEL
LIN {X 0,Y 270.213,Z 437.825,A -85,B 0,C 180,E1 -17797.037,E2 -17797.037} C_VEL
LIN {X 0,Y 270.304,Z 437.815,A -85,B 0,C 180,E1 -17800.245,E2 -17800.245} C_VEL
LIN {X 0,Y 270.406,Z 437.802,A -85,B 0,C 180,E1 -17804.936,E2 -17804.936} C_VEL
LIN {X 0,Y 270.416,Z 437.804,A -85,B 0,C 180,E1 -17809.518,E2 -17809.518} C_VEL
LIN {X 0,Y 270.589,Z 437.779,A -85,B 0,C 180,E1 -17812.538,E2 -17812.538} C_VEL
LIN {X 0,Y 270.791,Z 437.753,A -85,B 0,C 180,E1 -17818.513,E2 -17818.513} C_VEL
LIN {X 0,Y 270.791,Z 437.755,A -85,B 0,C 180,E1 -17821.487,E2 -17821.487} C_VEL
LIN {X 0,Y 270.588,Z 437.779,A -85,B 0,C 180,E1 -17827.462,E2 -17827.462} C_VEL
LIN {X 0,Y 270.416,Z 437.797,A -85,B 0,C 180,E1 -17830.482,E2 -17830.482} C_VEL
LIN {X 0,Y 270.406,Z 437.775,A -85,B 0,C 180,E1 -17835.065,E2 -17835.065} C_VEL
LIN {X 0,Y 270.304,Z 437.811,A -85,B 0,C 180,E1 -17839.755,E2 -17839.755} C_VEL
LIN {X 0,Y 270.276,Z 437.811,A -85,B 0,C 180,E1 -17844.586,E2 -17844.586} C_VEL
LIN {X 0,Y 270.272,Z 437.795,A -85,B 0,C 180,E1 -17847.909,E2 -17847.909} C_VEL
LIN {X 0,Y 270.186,Z 437.826,A -85,B 0,C 180,E1 -17851.348,E2 -17851.348} C_VEL
LIN {X 0,Y 270.204,Z 437.825,A -85,B 0,C 180,E1 -17854.905,E2 -17854.905} C_VEL
LIN {X 0,Y 270.2,Z 437.827,A -85,B 0,C 180,E1 -17858.71,E2 -17858.71} C_VEL
LIN {X 0,Y 270.191,Z 437.827,A -85,B 0,C 180,E1 -17863.254,E2 -17863.254} C_VEL
LIN {X 0,Y 270.251,Z 437.818,A -85,B 0,C 180,E1 -17867.457,E2 -17867.457} C_VEL
LIN {X 0,Y 270.247,Z 437.819,A -85,B 0,C 180,E1 -17871.381,E2 -17871.381} C_VEL
LIN {X 0,Y 270.219,Z 437.823,A -85,B 0,C 180,E1 -17875.097,E2 -17875.097} C_VEL
LIN {X 0,Y 270.203,Z 437.826,A -85,B 0,C 180,E1 -17879.131,E2 -17879.131} C_VEL
LIN {X 0,Y 270.311,Z 437.816,A -85,B 0,C 180,E1 -17883.691,E2 -17883.691} C_VEL
LIN {X 0,Y 271.407,Z 440.784,A -85,B 0,C 180,E1 -17884.06,E2 -17884.06} C_VEL
LIN {X 0,Y 275.751,Z 451.873,A -85,B 0,C 180,E1 -17885.584,E2 -17885.584} C_VEL
LIN {X 0,Y 279.147,Z 462.109,A -85,B 0,C 180,E1 -17887.177,E2 -17887.177} C_VEL
LIN {X 0,Y 281.196,Z 469.852,A -85,B 0,C 180,E1 -17888.523,E2 -17888.523} C_VEL
LIN {X 0,Y 279.588,Z 480.182,A -85,B 0,C 180,E1 -17890.163,E2 -17890.163} C_VEL
LIN {X 0,Y 278.013,Z 489.212,A -85,B 0,C 180,E1 -17891.96,E2 -17891.96} C_VEL
LIN {X 0,Y 276.119,Z 497.993,A -85,B 0,C 180,E1 -17894.12,E2 -17894.12} C_VEL
LIN {X 0,Y 274.607,Z 505.035,A -85,B 0,C 180,E1 -17896.306,E2 -17896.306} C_VEL
LIN {X 0,Y 273.588,Z 509.769,A -85,B 0,C 180,E1 -17898.141,E2 -17898.141} C_VEL
LIN {X 0,Y 272.56,Z 514.364,A -85,B 0,C 180,E1 -17900.351,E2 -17900.351} C_VEL
LIN {X 0,Y 271.639,Z 517.895,A -85,B 0,C 180,E1 -17902.567,E2 -17902.567} C_VEL
LIN {X 0,Y 271.176,Z 519.716,A -85,B 0,C 180,E1 -17904.049,E2 -17904.049} C_VEL
LIN {X 0,Y 270.806,Z 521.087,A -85,B 0,C 180,E1 -17905.534,E2 -17905.534} C_VEL
LIN {X 0,Y 270.715,Z 522.613,A -85,B 0,C 180,E1 -17908.512,E2 -17908.512} C_VEL
LIN {X 0,Y 270.692,Z 522.835,A -85,B 0,C 180,E1 -17910,E2 -17910} C_VEL
LIN {X 0,Y 270.715,Z 522.649,A -85,B 0,C 180,E1 -17911.488,E2 -17911.488} C_VEL
LIN {X 0,Y 270.797,Z 521.171,A -85,B 0,C 180,E1 -17914.465,E2 -17914.465} C_VEL
LIN {X 0,Y 271.162,Z 519.839,A -85,B 0,C 180,E1 -17915.951,E2 -17915.951} C_VEL
LIN {X 0,Y 271.948,Z 517.017,A -85,B 0,C 180,E1 -17918.171,E2 -17918.171} C_VEL
LIN {X 0,Y 272.922,Z 513.197,A -85,B 0,C 180,E1 -17920.385,E2 -17920.385} C_VEL
LIN {X 0,Y 274.079,Z 507.288,A -85,B 0,C 180,E1 -17922.99,E2 -17922.99} C_VEL
LIN {X 0,Y 275.584,Z 500.885,A -85,B 0,C 180,E1 -17925.153,E2 -17925.153} C_VEL
LIN {X 0,Y 277.331,Z 492.846,A -85,B 0,C 180,E1 -17927.323,E2 -17927.323} C_VEL
LIN {X 0,Y 278.803,Z 484.624,A -85,B 0,C 180,E1 -17929.129,E2 -17929.129} C_VEL
LIN {X 0,Y 280.476,Z 475.135,A -85,B 0,C 180,E1 -17930.8,E2 -17930.8} C_VEL
LIN {X 0,Y 281.129,Z 470.912,A -85,B 0,C 180,E1 -17931.443,E2 -17931.443} C_VEL
LIN {X 0,Y 281.047,Z 469.053,A -85,B 0,C 180,E1 -17931.74,E2 -17931.74} C_VEL
LIN {X 0,Y 277.987,Z 458.12,A -85,B 0,C 180,E1 -17933.585,E2 -17933.585} C_VEL
LIN {X 0,Y 274.039,Z 447.304,A -85,B 0,C 180,E1 -17935.196,E2 -17935.196} C_VEL
LIN {X 0,Y 270.397,Z 438.377,A -85,B 0,C 180,E1 -17936.378,E2 -17936.378} C_VEL
LIN {X 0,Y 270.31,Z 437.813,A -85,B 0,C 180,E1 -17936.439,E2 -17936.439} C_VEL
LIN {X 0,Y 270.202,Z 437.826,A -85,B 0,C 180,E1 -17940.869,E2 -17940.869} C_VEL
LIN {X 0,Y 270.218,Z 437.823,A -85,B 0,C 180,E1 -17944.903,E2 -17944.903} C_VEL
LIN {X 0,Y 270.254,Z 437.822,A -85,B 0,C 180,E1 -17948.725,E2 -17948.725} C_VEL
LIN {X 0,Y 270.25,Z 437.821,A -85,B 0,C 180,E1 -17952.543,E2 -17952.543} C_VEL
LIN {X 0,Y 270.19,Z 437.83,A -85,B 0,C 180,E1 -17956.745,E2 -17956.745} C_VEL
LIN {X 0,Y 270.208,Z 437.826,A -85,B 0,C 180,E1 -17961.374,E2 -17961.374} C_VEL
LIN {X 0,Y 270.203,Z 437.829,A -85,B 0,C 180,E1 -17965.094,E2 -17965.094} C_VEL
LIN {X 0,Y 270.202,Z 437.828,A -85,B 0,C 180,E1 -17969.13,E2 -17969.13} C_VEL
LIN {X 0,Y 270.265,Z 437.816,A -85,B 0,C 180,E1 -17972.146,E2 -17972.146} C_VEL
LIN {X 0,Y 270.279,Z 437.816,A -85,B 0,C 180,E1 -17975.519,E2 -17975.519} C_VEL
LIN {X 0,Y 270.304,Z 437.814,A -85,B 0,C 180,E1 -17980.244,E2 -17980.244} C_VEL
LIN {X 0,Y 270.405,Z 437.802,A -85,B 0,C 180,E1 -17984.935,E2 -17984.935} C_VEL
LIN {X 0,Y 270.415,Z 437.798,A -85,B 0,C 180,E1 -17989.518,E2 -17989.518} C_VEL
LIN {X 0,Y 270.588,Z 437.778,A -85,B 0,C 180,E1 -17992.538,E2 -17992.538} C_VEL
LIN {X 0,Y 270.79,Z 437.756,A -85,B 0,C 180,E1 -17998.513,E2 -17998.513} C_VEL
LIN {X 0,Y 270.79,Z 437.746,A -85,B 0,C 180,E1 -18001.487,E2 -18001.487} C_VEL
LIN {X 0,Y 270.587,Z 437.773,A -85,B 0,C 180,E1 -18007.462,E2 -18007.462} C_VEL
LIN {X 0,Y 270.414,Z 437.801,A -85,B 0,C 180,E1 -18010.482,E2 -18010.482} C_VEL
LIN {X 0,Y 270.405,Z 437.801,A -85,B 0,C 180,E1 -18015.064,E2 -18015.064} C_VEL
LIN {X 0,Y 270.303,Z 437.816,A -85,B 0,C 180,E1 -18019.755,E2 -18019.755} C_VEL
LIN {X 0,Y 270.206,Z 437.825,A -85,B 0,C 180,E1 -18023.105,E2 -18023.105} C_VEL
LIN {X 0,Y 269.517,Z 437.914,A -85,B 0,C 180,E1 -18024.35,E2 -18024.35} C_VEL
LIN {X 0,Y 266.653,Z 438.271,A -85,B 0,C 180,E1 -18026.378,E2 -18026.378} C_VEL
LIN {X 0,Y 264.237,Z 438.572,A -85,B 0,C 180,E1 -18028.026,E2 -18028.026} C_VEL
LIN {X 0,Y 263.205,Z 438.698,A -85,B 0,C 180,E1 -18029.305,E2 -18029.305} C_VEL
LIN {X 0,Y 263.122,Z 438.706,A -85,B 0,C 180,E1 -18029.738,E2 -18029.738} C_VEL
LIN {X 0,Y 263.174,Z 438.703,A -85,B 0,C 180,E1 -18034.122,E2 -18034.122} C_VEL
LIN {X 0,Y 263.222,Z 438.777,A -85,B 0,C 180,E1 -18036.775,E2 -18036.775} C_VEL
LIN {X 0,Y 264.405,Z 444.867,A -85,B 0,C 180,E1 -18040.634,E2 -18040.634} C_VEL
LIN {X 0,Y 265.687,Z 451.315,A -85,B 0,C 180,E1 -18044.421,E2 -18044.421} C_VEL
LIN {X 0,Y 267.075,Z 458.115,A -85,B 0,C 180,E1 -18048.204,E2 -18048.204} C_VEL
LIN {X 0,Y 267.824,Z 463.419,A -85,B 0,C 180,E1 -18050.966,E2 -18050.966} C_VEL
LIN {X 0,Y 266.879,Z 469.058,A -85,B 0,C 180,E1 -18053.664,E2 -18053.664} C_VEL
LIN {X 0,Y 265.1,Z 478.332,A -85,B 0,C 180,E1 -18058.032,E2 -18058.032} C_VEL
LIN {X 0,Y 263.861,Z 486.551,A -85,B 0,C 180,E1 -18061.887,E2 -18061.887} C_VEL
LIN {X 0,Y 266.305,Z 500.627,A -85,B 0,C 180,E1 -18062.808,E2 -18062.808} C_VEL
LIN {X 0,Y 267.773,Z 512.848,A -85,B 0,C 180,E1 -18063.825,E2 -18063.825} C_VEL
LIN {X 0,Y 268.535,Z 525.371,A -85,B 0,C 180,E1 -18065.105,E2 -18065.105} C_VEL
LIN {X 0,Y 268.52,Z 537.545,A -85,B 0,C 180,E1 -18066.62,E2 -18066.62} C_VEL
LIN {X 0,Y 268.058,Z 548.417,A -85,B 0,C 180,E1 -18068.264,E2 -18068.264} C_VEL
LIN {X 0,Y 267.104,Z 557.979,A -85,B 0,C 180,E1 -18069.998,E2 -18069.998} C_VEL
LIN {X 0,Y 265.455,Z 566.622,A -85,B 0,C 180,E1 -18071.876,E2 -18071.876} C_VEL
LIN {X 0,Y 263.809,Z 574.667,A -85,B 0,C 180,E1 -18074.027,E2 -18074.027} C_VEL
LIN {X 0,Y 262.791,Z 581.97,A -85,B 0,C 180,E1 -18076.467,E2 -18076.467} C_VEL
LIN {X 0,Y 262.085,Z 588.325,A -85,B 0,C 180,E1 -18079.181,E2 -18079.181} C_VEL
LIN {X 0,Y 261.975,Z 592.51,A -85,B 0,C 180,E1 -18081.515,E2 -18081.515} C_VEL
LIN {X 0,Y 262.153,Z 595.642,A -85,B 0,C 180,E1 -18083.844,E2 -18083.844} C_VEL
LIN {X 0,Y 262.436,Z 597.162,A -85,B 0,C 180,E1 -18085.392,E2 -18085.392} C_VEL
LIN {X 0,Y 262.659,Z 598.249,A -85,B 0,C 180,E1 -18086.933,E2 -18086.933} C_VEL
LIN {X 0,Y 263.254,Z 599.201,A -85,B 0,C 180,E1 -18090,E2 -18090} C_VEL
LIN {X 0,Y 262.659,Z 598.236,A -85,B 0,C 180,E1 -18093.068,E2 -18093.068} C_VEL
LIN {X 0,Y 262.434,Z 597.145,A -85,B 0,C 180,E1 -18094.608,E2 -18094.608} C_VEL
LIN {X 0,Y 262.076,Z 594.386,A -85,B 0,C 180,E1 -18097.153,E2 -18097.153} C_VEL
LIN {X 0,Y 261.988,Z 591.171,A -85,B 0,C 180,E1 -18099.262,E2 -18099.262} C_VEL
LIN {X 0,Y 262.214,Z 586.599,A -85,B 0,C 180,E1 -18101.597,E2 -18101.597} C_VEL
LIN {X 0,Y 262.917,Z 580.846,A -85,B 0,C 180,E1 -18103.921,E2 -18103.921} C_VEL
LIN {X 0,Y 264.093,Z 572.836,A -85,B 0,C 180,E1 -18106.481,E2 -18106.481} C_VEL
LIN {X 0,Y 265.456,Z 566.508,A -85,B 0,C 180,E1 -18108.125,E2 -18108.125} C_VEL
LIN {X 0,Y 267.09,Z 557.831,A -85,B 0,C 180,E1 -18110.003,E2 -18110.003} C_VEL
LIN {X 0,Y 268.019,Z 548.225,A -85,B 0,C 180,E1 -18111.74,E2 -18111.74} C_VEL
LIN {X 0,Y 268.526,Z 537.383,A -85,B 0,C 180,E1 -18113.371,E2 -18113.371} C_VEL
LIN {X 0,Y 268.48,Z 525.099,A -85,B 0,C 180,E1 -18114.897,E2 -18114.897} C_VEL
LIN {X 0,Y 267.69,Z 512.551,A -85,B 0,C 180,E1 -18116.172,E2 -18116.172} C_VEL
LIN {X 0,Y 266.098,Z 499.367,A -85,B 0,C 180,E1 -18117.249,E2 -18117.249} C_VEL
LIN {X 0,Y 263.841,Z 486.47,A -85,B 0,C 180,E1 -18118.11,E2 -18118.11} C_VEL
LIN {X 0,Y 265.427,Z 476.309,A -85,B 0,C 180,E1 -18122.875,E2 -18122.875} C_VEL
LIN {X 0,Y 266.841,Z 468.904,A -85,B 0,C 180,E1 -18126.342,E2 -18126.342} C_VEL
LIN {X 0,Y 267.857,Z 463.346,A -85,B 0,C 180,E1 -18129.029,E2 -18129.029} C_VEL
LIN {X 0,Y 267.055,Z 458.026,A -85,B 0,C 180,E1 -18131.795,E2 -18131.795} C_VEL
LIN {X 0,Y 265.674,Z 451.192,A -85,B 0,C 180,E1 -18135.582,E2 -18135.582} C_VEL
LIN {X 0,Y 264.129,Z 443.226,A -85,B 0,C 180,E1 -18140.313,E2 -18140.313} C_VEL
LIN {X 0,Y 263.223,Z 438.698,A -85,B 0,C 180,E1 -18143.226,E2 -18143.226} C_VEL
LIN {X 0,Y 263.186,Z 438.703,A -85,B 0,C 180,E1 -18145.891,E2 -18145.891} C_VEL
LIN {X 0,Y 263.143,Z 438.707,A -85,B 0,C 180,E1 -18149.506,E2 -18149.506} C_VEL
LIN {X 0,Y 263.193,Z 438.703,A -85,B 0,C 180,E1 -18153.003,E2 -18153.003} C_VEL
LIN {X 0,Y 263.158,Z 438.705,A -85,B 0,C 180,E1 -18156.385,E2 -18156.385} C_VEL
LIN {X 0,Y 263.265,Z 438.692,A -85,B 0,C 180,E1 -18159.694,E2 -18159.694} C_VEL
LIN {X 0,Y 263.354,Z 438.681,A -85,B 0,C 180,E1 -18164.522,E2 -18164.522} C_VEL
LIN {X 0,Y 263.358,Z 438.681,A -85,B 0,C 180,E1 -18169.234,E2 -18169.234} C_VEL
LIN {X 0,Y 263.548,Z 438.657,A -85,B 0,C 180,E1 -18172.338,E2 -18172.338} C_VEL
LIN {X 0,Y 263.756,Z 438.63,A -85,B 0,C 180,E1 -18178.473,E2 -18178.473} C_VEL
LIN {X 0,Y 263.755,Z 438.632,A -85,B 0,C 180,E1 -18181.527,E2 -18181.527} C_VEL
LIN {X 0,Y 263.547,Z 438.657,A -85,B 0,C 180,E1 -18187.662,E2 -18187.662} C_VEL
LIN {X 0,Y 263.358,Z 438.677,A -85,B 0,C 180,E1 -18190.766,E2 -18190.766} C_VEL
LIN {X 0,Y 263.354,Z 438.649,A -85,B 0,C 180,E1 -18195.478,E2 -18195.478} C_VEL
LIN {X 0,Y 263.267,Z 438.685,A -85,B 0,C 180,E1 -18200.307,E2 -18200.307} C_VEL
LIN {X 0,Y 263.21,Z 438.685,A -85,B 0,C 180,E1 -18205.291,E2 -18205.291} C_VEL
LIN {X 0,Y 263.168,Z 438.68,A -85,B 0,C 180,E1 -18208.731,E2 -18208.731} C_VEL
LIN {X 0,Y 263.135,Z 438.704,A -85,B 0,C 180,E1 -18212.288,E2 -18212.288} C_VEL
LIN {X 0,Y 263.184,Z 438.699,A -85,B 0,C 180,E1 -18216.763,E2 -18216.763} C_VEL
LIN {X 0,Y 263.132,Z 438.708,A -85,B 0,C 180,E1 -18221.595,E2 -18221.595} C_VEL
LIN {X 0,Y 263.147,Z 438.704,A -85,B 0,C 180,E1 -18226.021,E2 -18226.021} C_VEL
LIN {X 0,Y 263.213,Z 438.694,A -85,B 0,C 180,E1 -18228.385,E2 -18228.385} C_VEL
LIN {X 0,Y 263.21,Z 438.693,A -85,B 0,C 180,E1 -18233.229,E2 -18233.229} C_VEL
LIN {X 0,Y 263.186,Z 438.695,A -85,B 0,C 180,E1 -18235.89,E2 -18235.89} C_VEL
LIN {X 0,Y 263.153,Z 438.704,A -85,B 0,C 180,E1 -18239.507,E2 -18239.507} C_VEL
LIN {X 0,Y 263.292,Z 438.689,A -85,B 0,C 180,E1 -18242.919,E2 -18242.919} C_VEL
LIN {X 0,Y 263.88,Z 440.802,A -85,B 0,C 180,E1 -18243.162,E2 -18243.162} C_VEL
LIN {X 0,Y 267.667,Z 449.719,A -85,B 0,C 180,E1 -18244.427,E2 -18244.427} C_VEL
LIN {X 0,Y 271.218,Z 459.685,A -85,B 0,C 180,E1 -18245.984,E2 -18245.984} C_VEL
LIN {X 0,Y 274.13,Z 469.804,A -85,B 0,C 180,E1 -18247.758,E2 -18247.758} C_VEL
LIN {X 0,Y 274.556,Z 472.08,A -85,B 0,C 180,E1 -18248.168,E2 -18248.168} C_VEL
LIN {X 0,Y 272.994,Z 481.19,A -85,B 0,C 180,E1 -18249.662,E2 -18249.662} C_VEL
LIN {X 0,Y 271.34,Z 490.22,A -85,B 0,C 180,E1 -18251.501,E2 -18251.501} C_VEL
LIN {X 0,Y 269.367,Z 499.001,A -85,B 0,C 180,E1 -18253.711,E2 -18253.711} C_VEL
LIN {X 0,Y 267.784,Z 506.042,A -85,B 0,C 180,E1 -18255.95,E2 -18255.95} C_VEL
LIN {X 0,Y 266.714,Z 510.775,A -85,B 0,C 180,E1 -18257.83,E2 -18257.83} C_VEL
LIN {X 0,Y 265.635,Z 515.371,A -85,B 0,C 180,E1 -18260.097,E2 -18260.097} C_VEL
LIN {X 0,Y 264.672,Z 518.901,A -85,B 0,C 180,E1 -18262.37,E2 -18262.37} C_VEL
LIN {X 0,Y 264.187,Z 520.722,A -85,B 0,C 180,E1 -18263.891,E2 -18263.891} C_VEL
LIN {X 0,Y 263.8,Z 522.092,A -85,B 0,C 180,E1 -18265.416,E2 -18265.416} C_VEL
LIN {X 0,Y 263.692,Z 523.618,A -85,B 0,C 180,E1 -18268.473,E2 -18268.473} C_VEL
LIN {X 0,Y 263.667,Z 523.84,A -85,B 0,C 180,E1 -18270,E2 -18270} C_VEL
LIN {X 0,Y 263.691,Z 523.654,A -85,B 0,C 180,E1 -18271.527,E2 -18271.527} C_VEL
LIN {X 0,Y 263.79,Z 522.176,A -85,B 0,C 180,E1 -18274.584,E2 -18274.584} C_VEL
LIN {X 0,Y 264.172,Z 520.844,A -85,B 0,C 180,E1 -18276.109,E2 -18276.109} C_VEL
LIN {X 0,Y 264.994,Z 518.021,A -85,B 0,C 180,E1 -18278.387,E2 -18278.387} C_VEL
LIN {X 0,Y 266.012,Z 514.201,A -85,B 0,C 180,E1 -18280.657,E2 -18280.657} C_VEL
LIN {X 0,Y 267.242,Z 508.276,A -85,B 0,C 180,E1 -18283.334,E2 -18283.334} C_VEL
LIN {X 0,Y 269.074,Z 500.689,A -85,B 0,C 180,E1 -18285.917,E2 -18285.917} C_VEL
LIN {X 0,Y 270.929,Z 492.32,A -85,B 0,C 180,E1 -18288.137,E2 -18288.137} C_VEL
LIN {X 0,Y 272.507,Z 483.733,A -85,B 0,C 180,E1 -18289.982,E2 -18289.982} C_VEL
LIN {X 0,Y 274.293,Z 473.699,A -85,B 0,C 180,E1 -18291.709,E2 -18291.709} C_VEL
LIN {X 0,Y 274.529,Z 471.924,A -85,B 0,C 180,E1 -18291.985,E2 -18291.985} C_VEL
LIN {X 0,Y 272.23,Z 462.813,A -85,B 0,C 180,E1 -18293.613,E2 -18293.613} C_VEL
LIN {X 0,Y 269.321,Z 454.124,A -85,B 0,C 180,E1 -18295.034,E2 -18295.034} C_VEL
LIN {X 0,Y 265.583,Z 444.511,A -85,B 0,C 180,E1 -18296.45,E2 -18296.45} C_VEL
LIN {X 0,Y 263.281,Z 438.877,A -85,B 0,C 180,E1 -18297.194,E2 -18297.194} C_VEL
LIN {X 0,Y 263.142,Z 438.704,A -85,B 0,C 180,E1 -18301.278,E2 -18301.278} C_VEL
LIN {X 0,Y 263.175,Z 438.7,A -85,B 0,C 180,E1 -18304.122,E2 -18304.122} C_VEL
LIN {X 0,Y 263.191,Z 438.7,A -85,B 0,C 180,E1 -18307.892,E2 -18307.892} C_VEL
LIN {X 0,Y 263.208,Z 438.697,A -85,B 0,C 180,E1 -18311.877,E2 -18311.877} C_VEL
LIN {X 0,Y 263.14,Z 438.706,A -85,B 0,C 180,E1 -18316.147,E2 -18316.147} C_VEL
LIN {X 0,Y 263.109,Z 438.71,A -85,B 0,C 180,E1 -18320.128,E2 -18320.128} C_VEL
LIN {X 0,Y 263.164,Z 438.701,A -85,B 0,C 180,E1 -18324.018,E2 -18324.018} C_VEL
LIN {X 0,Y 263.134,Z 438.703,A -85,B 0,C 180,E1 -18327.712,E2 -18327.712} C_VEL
LIN {X 0,Y 263.197,Z 438.696,A -85,B 0,C 180,E1 -18331.785,E2 -18331.785} C_VEL
LIN {X 0,Y 263.227,Z 438.696,A -85,B 0,C 180,E1 -18335.2,E2 -18335.2} C_VEL
LIN {X 0,Y 263.265,Z 438.69,A -85,B 0,C 180,E1 -18339.693,E2 -18339.693} C_VEL
LIN {X 0,Y 263.353,Z 438.68,A -85,B 0,C 180,E1 -18344.522,E2 -18344.522} C_VEL
LIN {X 0,Y 263.357,Z 438.677,A -85,B 0,C 180,E1 -18349.234,E2 -18349.234} C_VEL
LIN {X 0,Y 263.547,Z 438.657,A -85,B 0,C 180,E1 -18352.338,E2 -18352.338} C_VEL
LIN {X 0,Y 263.754,Z 438.632,A -85,B 0,C 180,E1 -18358.473,E2 -18358.473} C_VEL
LIN {X 0,Y 263.754,Z 438.622,A -85,B 0,C 180,E1 -18361.527,E2 -18361.527} C_VEL
LIN {X 0,Y 263.546,Z 438.65,A -85,B 0,C 180,E1 -18367.662,E2 -18367.662} C_VEL
LIN {X 0,Y 263.357,Z 438.679,A -85,B 0,C 180,E1 -18370.766,E2 -18370.766} C_VEL
LIN {X 0,Y 263.353,Z 438.679,A -85,B 0,C 180,E1 -18375.478,E2 -18375.478} C_VEL
LIN {X 0,Y 263.264,Z 438.694,A -85,B 0,C 180,E1 -18380.307,E2 -18380.307} C_VEL
LIN {X 0,Y 263.194,Z 438.7,A -85,B 0,C 180,E1 -18385.293,E2 -18385.293} C_VEL
LIN {X 0,Y 263.167,Z 438.703,A -85,B 0,C 180,E1 -18388.731,E2 -18388.731} C_VEL
LIN {X 0,Y 263.122,Z 438.706,A -85,B 0,C 180,E1 -18389.738,E2 -18389.738} C_VEL
LIN {X 0,Y 262.442,Z 438.796,A -85,B 0,C 180,E1 -18390.589,E2 -18390.589} C_VEL
LIN {X 0,Y 259.591,Z 439.15,A -85,B 0,C 180,E1 -18391.923,E2 -18391.923} C_VEL
LIN {X 0,Y 256.742,Z 439.506,A -85,B 0,C 180,E1 -18393.286,E2 -18393.286} C_VEL
LIN {X 0,Y 256.098,Z 439.584,A -85,B 0,C 180,E1 -18394.169,E2 -18394.169} C_VEL
LIN {X 0,Y 256.161,Z 439.644,A -85,B 0,C 180,E1 -18396.026,E2 -18396.026} C_VEL
LIN {X 0,Y 257.389,Z 445.88,A -85,B 0,C 180,E1 -18400.134,E2 -18400.134} C_VEL
LIN {X 0,Y 258.614,Z 451.978,A -85,B 0,C 180,E1 -18403.866,E2 -18403.866} C_VEL
LIN {X 0,Y 259.851,Z 458.236,A -85,B 0,C 180,E1 -18407.456,E2 -18407.456} C_VEL
LIN {X 0,Y 260.837,Z 464.124,A -85,B 0,C 180,E1 -18410.658,E2 -18410.658} C_VEL
LIN {X 0,Y 260.25,Z 468.001,A -85,B 0,C 180,E1 -18412.583,E2 -18412.583} C_VEL
LIN {X 0,Y 258.414,Z 477.177,A -85,B 0,C 180,E1 -18417.048,E2 -18417.048} C_VEL
LIN {X 0,Y 257.012,Z 485.542,A -85,B 0,C 180,E1 -18421.071,E2 -18421.071} C_VEL
LIN {X 0,Y 259.565,Z 499.774,A -85,B 0,C 180,E1 -18422.054,E2 -18422.054} C_VEL
LIN {X 0,Y 261.013,Z 511.775,A -85,B 0,C 180,E1 -18423.093,E2 -18423.093} C_VEL
LIN {X 0,Y 261.767,Z 524.416,A -85,B 0,C 180,E1 -18424.429,E2 -18424.429} C_VEL
LIN {X 0,Y 261.776,Z 535.91,A -85,B 0,C 180,E1 -18425.897,E2 -18425.897} C_VEL
LIN {X 0,Y 261.263,Z 547.372,A -85,B 0,C 180,E1 -18427.669,E2 -18427.669} C_VEL
LIN {X 0,Y 260.349,Z 556.952,A -85,B 0,C 180,E1 -18429.456,E2 -18429.456} C_VEL
LIN {X 0,Y 258.633,Z 565.595,A -85,B 0,C 180,E1 -18431.38,E2 -18431.38} C_VEL
LIN {X 0,Y 257.078,Z 572.665,A -85,B 0,C 180,E1 -18433.284,E2 -18433.284} C_VEL
LIN {X 0,Y 255.969,Z 579.897,A -85,B 0,C 180,E1 -18435.694,E2 -18435.694} C_VEL
LIN {X 0,Y 255.191,Z 585.635,A -85,B 0,C 180,E1 -18438.08,E2 -18438.08} C_VEL
LIN {X 0,Y 254.917,Z 590.192,A -85,B 0,C 180,E1 -18440.479,E2 -18440.479} C_VEL
LIN {X 0,Y 255.015,Z 593.591,A -85,B 0,C 180,E1 -18442.809,E2 -18442.809} C_VEL
LIN {X 0,Y 255.359,Z 596.147,A -85,B 0,C 180,E1 -18445.264,E2 -18445.264} C_VEL
LIN {X 0,Y 255.595,Z 597.237,A -85,B 0,C 180,E1 -18446.848,E2 -18446.848} C_VEL
LIN {X 0,Y 256.22,Z 598.195,A -85,B 0,C 180,E1 -18450,E2 -18450} C_VEL
LIN {X 0,Y 255.595,Z 597.224,A -85,B 0,C 180,E1 -18453.153,E2 -18453.153} C_VEL
LIN {X 0,Y 255.357,Z 596.129,A -85,B 0,C 180,E1 -18454.736,E2 -18454.736} C_VEL
LIN {X 0,Y 255.025,Z 593.54,A -85,B 0,C 180,E1 -18457.21,E2 -18457.21} C_VEL
LIN {X 0,Y 254.918,Z 590.145,A -85,B 0,C 180,E1 -18459.522,E2 -18459.522} C_VEL
LIN {X 0,Y 255.191,Z 585.572,A -85,B 0,C 180,E1 -18461.92,E2 -18461.92} C_VEL
LIN {X 0,Y 255.967,Z 579.819,A -85,B 0,C 180,E1 -18464.307,E2 -18464.307} C_VEL
LIN {X 0,Y 257.082,Z 572.557,A -85,B 0,C 180,E1 -18466.719,E2 -18466.719} C_VEL
LIN {X 0,Y 258.633,Z 565.477,A -85,B 0,C 180,E1 -18468.62,E2 -18468.62} C_VEL
LIN {X 0,Y 260.462,Z 555.797,A -85,B 0,C 180,E1 -18470.742,E2 -18470.742} C_VEL
LIN {X 0,Y 261.407,Z 544.751,A -85,B 0,C 180,E1 -18472.736,E2 -18472.736} C_VEL
LIN {X 0,Y 261.819,Z 533.902,A -85,B 0,C 180,E1 -18474.352,E2 -18474.352} C_VEL
LIN {X 0,Y 261.587,Z 521.787,A -85,B 0,C 180,E1 -18475.843,E2 -18475.843} C_VEL
LIN {X 0,Y 260.664,Z 508.65,A -85,B 0,C 180,E1 -18477.159,E2 -18477.159} C_VEL
LIN {X 0,Y 258.778,Z 495.016,A -85,B 0,C 180,E1 -18478.272,E2 -18478.272} C_VEL
LIN {X 0,Y 256.996,Z 485.34,A -85,B 0,C 180,E1 -18478.944,E2 -18478.944} C_VEL
LIN {X 0,Y 258.761,Z 475.258,A -85,B 0,C 180,E1 -18483.834,E2 -18483.834} C_VEL
LIN {X 0,Y 260.717,Z 465.538,A -85,B 0,C 180,E1 -18488.58,E2 -18488.58} C_VEL
LIN {X 0,Y 260.848,Z 464.038,A -85,B 0,C 180,E1 -18489.34,E2 -18489.34} C_VEL
LIN {X 0,Y 259.657,Z 457.208,A -85,B 0,C 180,E1 -18493.047,E2 -18493.047} C_VEL
LIN {X 0,Y 258.194,Z 449.935,A -85,B 0,C 180,E1 -18497.302,E2 -18497.302} C_VEL
LIN {X 0,Y 257.044,Z 443.939,A -85,B 0,C 180,E1 -18501.034,E2 -18501.034} C_VEL
LIN {X 0,Y 256.139,Z 439.581,A -85,B 0,C 180,E1 -18504.091,E2 -18504.091} C_VEL
LIN {X 0,Y 256.095,Z 439.583,A -85,B 0,C 180,E1 -18508.573,E2 -18508.573} C_VEL
LIN {X 0,Y 256.14,Z 439.582,A -85,B 0,C 180,E1 -18512.196,E2 -18512.196} C_VEL
LIN {X 0,Y 256.145,Z 439.579,A -85,B 0,C 180,E1 -18515.697,E2 -18515.697} C_VEL
LIN {X 0,Y 256.165,Z 439.574,A -85,B 0,C 180,E1 -18519.105,E2 -18519.105} C_VEL
LIN {X 0,Y 256.303,Z 439.562,A -85,B 0,C 180,E1 -18524.085,E2 -18524.085} C_VEL
LIN {X 0,Y 256.299,Z 439.562,A -85,B 0,C 180,E1 -18527.328,E2 -18527.328} C_VEL
LIN {X 0,Y 256.508,Z 439.535,A -85,B 0,C 180,E1 -18532.126,E2 -18532.126} C_VEL
LIN {X 0,Y 256.504,Z 439.532,A -85,B 0,C 180,E1 -18536.859,E2 -18536.859} C_VEL
LIN {X 0,Y 256.777,Z 439.499,A -85,B 0,C 180,E1 -18540,E2 -18540} C_VEL
LIN {X 0,Y 256.502,Z 439.534,A -85,B 0,C 180,E1 -18543.141,E2 -18543.141} C_VEL
LIN {X 0,Y 256.507,Z 439.534,A -85,B 0,C 180,E1 -18547.874,E2 -18547.874} C_VEL
LIN {X 0,Y 256.299,Z 439.548,A -85,B 0,C 180,E1 -18552.672,E2 -18552.672} C_VEL
LIN {X 0,Y 256.285,Z 439.528,A -85,B 0,C 180,E1 -18556.302,E2 -18556.302} C_VEL
LIN {X 0,Y 256.161,Z 439.573,A -85,B 0,C 180,E1 -18561.12,E2 -18561.12} C_VEL
LIN {X 0,Y 256.191,Z 439.56,A -85,B 0,C 180,E1 -18565.138,E2 -18565.138} C_VEL
LIN {X 0,Y 256.106,Z 439.566,A -85,B 0,C 180,E1 -18569.601,E2 -18569.601} C_VEL
LIN {X 0,Y 256.07,Z 439.588,A -85,B 0,C 180,E1 -18573.293,E2 -18573.293} C_VEL
LIN {X 0,Y 256.117,Z 439.583,A -85,B 0,C 180,E1 -18577.271,E2 -18577.271} C_VEL
LIN {X 0,Y 256.062,Z 439.59,A -85,B 0,C 180,E1 -18581.202,E2 -18581.202} C_VEL
LIN {X 0,Y 256.078,Z 439.586,A -85,B 0,C 180,E1 -18585.526,E2 -18585.526} C_VEL
LIN {X 0,Y 256.134,Z 439.578,A -85,B 0,C 180,E1 -18588.812,E2 -18588.812} C_VEL
LIN {X 0,Y 256.159,Z 439.573,A -85,B 0,C 180,E1 -18592.872,E2 -18592.872} C_VEL
LIN {X 0,Y 256.088,Z 439.581,A -85,B 0,C 180,E1 -18596.71,E2 -18596.71} C_VEL
LIN {X 0,Y 256.14,Z 439.58,A -85,B 0,C 180,E1 -18601.405,E2 -18601.405} C_VEL
LIN {X 0,Y 256.209,Z 439.614,A -85,B 0,C 180,E1 -18602.095,E2 -18602.095} C_VEL
LIN {X 0,Y 256.987,Z 441.964,A -85,B 0,C 180,E1 -18602.385,E2 -18602.385} C_VEL
LIN {X 0,Y 261.441,Z 452.432,A -85,B 0,C 180,E1 -18603.962,E2 -18603.962} C_VEL
LIN {X 0,Y 265.261,Z 463.568,A -85,B 0,C 180,E1 -18605.811,E2 -18605.811} C_VEL
LIN {X 0,Y 267.71,Z 472.462,A -85,B 0,C 180,E1 -18607.468,E2 -18607.468} C_VEL
LIN {X 0,Y 267.939,Z 473.737,A -85,B 0,C 180,E1 -18607.707,E2 -18607.707} C_VEL
LIN {X 0,Y 266.037,Z 484.128,A -85,B 0,C 180,E1 -18609.511,E2 -18609.511} C_VEL
LIN {X 0,Y 264.328,Z 492.822,A -85,B 0,C 180,E1 -18611.394,E2 -18611.394} C_VEL
LIN {X 0,Y 262.33,Z 501.317,A -85,B 0,C 180,E1 -18613.662,E2 -18613.662} C_VEL
LIN {X 0,Y 260.596,Z 508.525,A -85,B 0,C 180,E1 -18616.141,E2 -18616.141} C_VEL
LIN {X 0,Y 259.498,Z 513.432,A -85,B 0,C 180,E1 -18618.28,E2 -18618.28} C_VEL
LIN {X 0,Y 258.307,Z 517.672,A -85,B 0,C 180,E1 -18620.604,E2 -18620.604} C_VEL
LIN {X 0,Y 257.708,Z 519.907,A -85,B 0,C 180,E1 -18622.163,E2 -18622.163} C_VEL
LIN {X 0,Y 257.2,Z 521.728,A -85,B 0,C 180,E1 -18623.725,E2 -18623.725} C_VEL
LIN {X 0,Y 256.795,Z 523.098,A -85,B 0,C 180,E1 -18625.29,E2 -18625.29} C_VEL
LIN {X 0,Y 256.668,Z 524.623,A -85,B 0,C 180,E1 -18628.431,E2 -18628.431} C_VEL
LIN {X 0,Y 256.642,Z 524.845,A -85,B 0,C 180,E1 -18630,E2 -18630} C_VEL
LIN {X 0,Y 256.667,Z 524.659,A -85,B 0,C 180,E1 -18631.569,E2 -18631.569} C_VEL
LIN {X 0,Y 256.785,Z 523.181,A -85,B 0,C 180,E1 -18634.71,E2 -18634.71} C_VEL
LIN {X 0,Y 257.185,Z 521.848,A -85,B 0,C 180,E1 -18636.275,E2 -18636.275} C_VEL
LIN {X 0,Y 258.044,Z 519.025,A -85,B 0,C 180,E1 -18638.615,E2 -18638.615} C_VEL
LIN {X 0,Y 259.109,Z 515.205,A -85,B 0,C 180,E1 -18640.945,E2 -18640.945} C_VEL
LIN {X 0,Y 260.409,Z 509.278,A -85,B 0,C 180,E1 -18643.691,E2 -18643.691} C_VEL
LIN {X 0,Y 262.322,Z 501.692,A -85,B 0,C 180,E1 -18646.338,E2 -18646.338} C_VEL
LIN {X 0,Y 264.26,Z 493.322,A -85,B 0,C 180,E1 -18648.611,E2 -18648.611} C_VEL
LIN {X 0,Y 265.916,Z 484.734,A -85,B 0,C 180,E1 -18650.499,E2 -18650.499} C_VEL
LIN {X 0,Y 267.901,Z 474.106,A -85,B 0,C 180,E1 -18652.358,E2 -18652.358} C_VEL
LIN {X 0,Y 265.637,Z 464.547,A -85,B 0,C 180,E1 -18654.139,E2 -18654.139} C_VEL
LIN {X 0,Y 261.971,Z 453.901,A -85,B 0,C 180,E1 -18655.941,E2 -18655.941} C_VEL
LIN {X 0,Y 258.07,Z 444.331,A -85,B 0,C 180,E1 -18657.402,E2 -18657.402} C_VEL
LIN {X 0,Y 256.218,Z 439.776,A -85,B 0,C 180,E1 -18658.026,E2 -18658.026} C_VEL
LIN {X 0,Y 256.128,Z 439.567,A -85,B 0,C 180,E1 -18658.59,E2 -18658.59} C_VEL
LIN {X 0,Y 256.087,Z 439.586,A -85,B 0,C 180,E1 -18663.29,E2 -18663.29} C_VEL
LIN {X 0,Y 256.144,Z 439.58,A -85,B 0,C 180,E1 -18667.279,E2 -18667.279} C_VEL
LIN {X 0,Y 256.16,Z 439.578,A -85,B 0,C 180,E1 -18671.183,E2 -18671.183} C_VEL
LIN {X 0,Y 256.074,Z 439.587,A -85,B 0,C 180,E1 -18675.527,E2 -18675.527} C_VEL
LIN {X 0,Y 256.06,Z 439.587,A -85,B 0,C 180,E1 -18678.797,E2 -18678.797} C_VEL
LIN {X 0,Y 256.131,Z 439.578,A -85,B 0,C 180,E1 -18682.867,E2 -18682.867} C_VEL
LIN {X 0,Y 256.069,Z 439.587,A -85,B 0,C 180,E1 -18686.707,E2 -18686.707} C_VEL
LIN {X 0,Y 256.105,Z 439.584,A -85,B 0,C 180,E1 -18690.399,E2 -18690.399} C_VEL
LIN {X 0,Y 256.19,Z 439.575,A -85,B 0,C 180,E1 -18694.862,E2 -18694.862} C_VEL
LIN {X 0,Y 256.169,Z 439.575,A -85,B 0,C 180,E1 -18699.105,E2 -18699.105} C_VEL
LIN {X 0,Y 256.302,Z 439.555,A -85,B 0,C 180,E1 -18704.085,E2 -18704.085} C_VEL
LIN {X 0,Y 256.298,Z 439.555,A -85,B 0,C 180,E1 -18707.328,E2 -18707.328} C_VEL
LIN {X 0,Y 256.507,Z 439.533,A -85,B 0,C 180,E1 -18712.126,E2 -18712.126} C_VEL
LIN {X 0,Y 256.502,Z 439.533,A -85,B 0,C 180,E1 -18716.859,E2 -18716.859} C_VEL
LIN {X 0,Y 256.776,Z 439.499,A -85,B 0,C 180,E1 -18720,E2 -18720} C_VEL
LIN {X 0,Y 256.502,Z 439.53,A -85,B 0,C 180,E1 -18723.141,E2 -18723.141} C_VEL
LIN {X 0,Y 256.506,Z 439.527,A -85,B 0,C 180,E1 -18727.874,E2 -18727.874} C_VEL
LIN {X 0,Y 256.298,Z 439.555,A -85,B 0,C 180,E1 -18732.672,E2 -18732.672} C_VEL
LIN {X 0,Y 256.285,Z 439.559,A -85,B 0,C 180,E1 -18736.302,E2 -18736.302} C_VEL
LIN {X 0,Y 256.155,Z 439.577,A -85,B 0,C 180,E1 -18741.118,E2 -18741.118} C_VEL
LIN {X 0,Y 256.172,Z 439.575,A -85,B 0,C 180,E1 -18745.13,E2 -18745.13} C_VEL
LIN {X 0,Y 256.105,Z 439.582,A -85,B 0,C 180,E1 -18749.601,E2 -18749.601} C_VEL
LIN {X 0,Y 256.098,Z 439.584,A -85,B 0,C 180,E1 -18754.169,E2 -18754.169} C_VEL
LIN {X 0,Y 255.589,Z 440.153,A -85,B 0,C 180,E1 -18755.472,E2 -18755.472} C_VEL
LIN {X 0,Y 254.321,Z 441.601,A -85,B 0,C 180,E1 -18756.733,E2 -18756.733} C_VEL
LIN {X 0,Y 251.425,Z 445.948,A -85,B 0,C 180,E1 -18759.201,E2 -18759.201} C_VEL
LIN {X 0,Y 250.767,Z 448.186,A -85,B 0,C 180,E1 -18760.469,E2 -18760.469} C_VEL
LIN {X 0,Y 250.792,Z 448.885,A -85,B 0,C 180,E1 -18760.899,E2 -18760.899} C_VEL
LIN {X 0,Y 252.086,Z 455.625,A -85,B 0,C 180,E1 -18765.065,E2 -18765.065} C_VEL
LIN {X 0,Y 253.264,Z 461.593,A -85,B 0,C 180,E1 -18768.525,E2 -18768.525} C_VEL
LIN {X 0,Y 253.789,Z 465.777,A -85,B 0,C 180,E1 -18770.84,E2 -18770.84} C_VEL
LIN {X 0,Y 252.63,Z 471.561,A -85,B 0,C 180,E1 -18773.781,E2 -18773.781} C_VEL
LIN {X 0,Y 250.977,Z 479.7,A -85,B 0,C 180,E1 -18777.856,E2 -18777.856} C_VEL
LIN {X 0,Y 250.192,Z 484.344,A -85,B 0,C 180,E1 -18780.191,E2 -18780.191} C_VEL
LIN {X 0,Y 252.838,Z 498.792,A -85,B 0,C 180,E1 -18781.248,E2 -18781.248} C_VEL
LIN {X 0,Y 254.372,Z 512.104,A -85,B 0,C 180,E1 -18782.46,E2 -18782.46} C_VEL
LIN {X 0,Y 255.079,Z 525.484,A -85,B 0,C 180,E1 -18783.964,E2 -18783.964} C_VEL
LIN {X 0,Y 254.95,Z 537.341,A -85,B 0,C 180,E1 -18785.576,E2 -18785.576} C_VEL
LIN {X 0,Y 254.311,Z 548.605,A -85,B 0,C 180,E1 -18787.453,E2 -18787.453} C_VEL
LIN {X 0,Y 253.291,Z 557.764,A -85,B 0,C 180,E1 -18789.282,E2 -18789.282} C_VEL
LIN {X 0,Y 251.252,Z 567.621,A -85,B 0,C 180,E1 -18791.658,E2 -18791.658} C_VEL
LIN {X 0,Y 249.738,Z 574.294,A -85,B 0,C 180,E1 -18793.655,E2 -18793.655} C_VEL
LIN {X 0,Y 248.717,Z 580.956,A -85,B 0,C 180,E1 -18796.103,E2 -18796.103} C_VEL
LIN {X 0,Y 248.016,Z 586.276,A -85,B 0,C 180,E1 -18798.559,E2 -18798.559} C_VEL
LIN {X 0,Y 247.847,Z 590.468,A -85,B 0,C 180,E1 -18801.028,E2 -18801.028} C_VEL
LIN {X 0,Y 248.011,Z 593.608,A -85,B 0,C 180,E1 -18803.492,E2 -18803.492} C_VEL
LIN {X 0,Y 248.285,Z 595.132,A -85,B 0,C 180,E1 -18805.129,E2 -18805.129} C_VEL
LIN {X 0,Y 248.532,Z 596.226,A -85,B 0,C 180,E1 -18806.758,E2 -18806.758} C_VEL
LIN {X 0,Y 249.186,Z 597.189,A -85,B 0,C 180,E1 -18810,E2 -18810} C_VEL
LIN {X 0,Y 248.532,Z 596.212,A -85,B 0,C 180,E1 -18813.242,E2 -18813.242} C_VEL
LIN {X 0,Y 248.284,Z 595.113,A -85,B 0,C 180,E1 -18814.872,E2 -18814.872} C_VEL
LIN {X 0,Y 247.955,Z 592.731,A -85,B 0,C 180,E1 -18817.236,E2 -18817.236} C_VEL
LIN {X 0,Y 247.875,Z 589.123,A -85,B 0,C 180,E1 -18819.795,E2 -18819.795} C_VEL
LIN {X 0,Y 248.188,Z 584.546,A -85,B 0,C 180,E1 -18822.262,E2 -18822.262} C_VEL
LIN {X 0,Y 248.98,Z 578.786,A -85,B 0,C 180,E1 -18824.717,E2 -18824.717} C_VEL
LIN {X 0,Y 250.079,Z 572.227,A -85,B 0,C 180,E1 -18826.971,E2 -18826.971} C_VEL
LIN {X 0,Y 251.849,Z 564.45,A -85,B 0,C 180,E1 -18829.141,E2 -18829.141} C_VEL
LIN {X 0,Y 253.561,Z 555.759,A -85,B 0,C 180,E1 -18831.12,E2 -18831.12} C_VEL
LIN {X 0,Y 254.531,Z 544.906,A -85,B 0,C 180,E1 -18833.17,E2 -18833.17} C_VEL
LIN {X 0,Y 255.054,Z 534.16,A -85,B 0,C 180,E1 -18834.847,E2 -18834.847} C_VEL
LIN {X 0,Y 254.917,Z 522.203,A -85,B 0,C 180,E1 -18836.408,E2 -18836.408} C_VEL
LIN {X 0,Y 254.116,Z 509.634,A -85,B 0,C 180,E1 -18837.747,E2 -18837.747} C_VEL
LIN {X 0,Y 252.365,Z 496.468,A -85,B 0,C 180,E1 -18838.907,E2 -18838.907} C_VEL
LIN {X 0,Y 250.176,Z 484.297,A -85,B 0,C 180,E1 -18839.793,E2 -18839.793} C_VEL
LIN {X 0,Y 252.096,Z 474.195,A -85,B 0,C 180,E1 -18844.856,E2 -18844.856} C_VEL
LIN {X 0,Y 253.58,Z 467.181,A -85,B 0,C 180,E1 -18848.381,E2 -18848.381} C_VEL
LIN {X 0,Y 253.809,Z 464.896,A -85,B 0,C 180,E1 -18849.559,E2 -18849.559} C_VEL
LIN {X 0,Y 252.853,Z 459.291,A -85,B 0,C 180,E1 -18852.723,E2 -18852.723} C_VEL
LIN {X 0,Y 251.548,Z 452.773,A -85,B 0,C 180,E1 -18856.587,E2 -18856.587} C_VEL
LIN {X 0,Y 250.246,Z 446.14,A -85,B 0,C 180,E1 -18860.81,E2 -18860.81} C_VEL
LIN {X 0,Y 249.104,Z 440.455,A -85,B 0,C 180,E1 -18864.814,E2 -18864.814} C_VEL
LIN {X 0,Y 249.05,Z 440.462,A -85,B 0,C 180,E1 -18869.473,E2 -18869.473} C_VEL
LIN {X 0,Y 249.071,Z 440.463,A -85,B 0,C 180,E1 -18873.162,E2 -18873.162} C_VEL
LIN {X 0,Y 249.064,Z 440.46,A -85,B 0,C 180,E1 -18876.731,E2 -18876.731} C_VEL
LIN {X 0,Y 249.112,Z 440.455,A -85,B 0,C 180,E1 -18880.212,E2 -18880.212} C_VEL
LIN {X 0,Y 249.245,Z 440.44,A -85,B 0,C 180,E1 -18883.622,E2 -18883.622} C_VEL
LIN {X 0,Y 249.248,Z 440.438,A -85,B 0,C 180,E1 -18888.616,E2 -18888.616} C_VEL
LIN {X 0,Y 249.449,Z 440.416,A -85,B 0,C 180,E1 -18891.902,E2 -18891.902} C_VEL
LIN {X 0,Y 249.301,Z 440.432,A -85,B 0,C 180,E1 -18895.149,E2 -18895.149} C_VEL
LIN {X 0,Y 249.68,Z 440.383,A -85,B 0,C 180,E1 -18898.387,E2 -18898.387} C_VEL
LIN {X 0,Y 249.679,Z 440.386,A -85,B 0,C 180,E1 -18901.613,E2 -18901.613} C_VEL
LIN {X 0,Y 249.438,Z 440.41,A -85,B 0,C 180,E1 -18906.698,E2 -18906.698} C_VEL
LIN {X 0,Y 249.346,Z 440.424,A -85,B 0,C 180,E1 -18909.736,E2 -18909.736} C_VEL
LIN {X 0,Y 249.209,Z 440.41,A -85,B 0,C 180,E1 -18914.703,E2 -18914.703} C_VEL
LIN {X 0,Y 249.143,Z 440.431,A -85,B 0,C 180,E1 -18918.077,E2 -18918.077} C_VEL
LIN {X 0,Y 249.09,Z 440.457,A -85,B 0,C 180,E1 -18921.518,E2 -18921.518} C_VEL
LIN {X 0,Y 249.133,Z 440.434,A -85,B 0,C 180,E1 -18925.482,E2 -18925.482} C_VEL
LIN {X 0,Y 249.075,Z 440.434,A -85,B 0,C 180,E1 -18928.989,E2 -18928.989} C_VEL
LIN {X 0,Y 249.033,Z 440.461,A -85,B 0,C 180,E1 -18932.426,E2 -18932.426} C_VEL
LIN {X 0,Y 249.032,Z 440.46,A -85,B 0,C 180,E1 -18936.345,E2 -18936.345} C_VEL
LIN {X 0,Y 249.01,Z 440.463,A -85,B 0,C 180,E1 -18940.478,E2 -18940.478} C_VEL
LIN {X 0,Y 249.021,Z 440.464,A -85,B 0,C 180,E1 -18944.875,E2 -18944.875} C_VEL
LIN {X 0,Y 249.084,Z 440.454,A -85,B 0,C 180,E1 -18947.377,E2 -18947.377} C_VEL
LIN {X 0,Y 249.056,Z 440.458,A -85,B 0,C 180,E1 -18951.624,E2 -18951.624} C_VEL
LIN {X 0,Y 249.064,Z 440.454,A -85,B 0,C 180,E1 -18955.642,E2 -18955.642} C_VEL
LIN {X 0,Y 249.054,Z 440.461,A -85,B 0,C 180,E1 -18959.473,E2 -18959.473} C_VEL
LIN {X 0,Y 249.111,Z 440.537,A -85,B 0,C 180,E1 -18961.209,E2 -18961.209} C_VEL
LIN {X 0,Y 250.073,Z 443.227,A -85,B 0,C 180,E1 -18961.565,E2 -18961.565} C_VEL
LIN {X 0,Y 254.46,Z 453.124,A -85,B 0,C 180,E1 -18963.142,E2 -18963.142} C_VEL
LIN {X 0,Y 258.353,Z 464.365,A -85,B 0,C 180,E1 -18965.08,E2 -18965.08} C_VEL
LIN {X 0,Y 260.926,Z 473.719,A -85,B 0,C 180,E1 -18966.882,E2 -18966.882} C_VEL
LIN {X 0,Y 261.31,Z 475.384,A -85,B 0,C 180,E1 -18967.225,E2 -18967.225} C_VEL
LIN {X 0,Y 259.471,Z 485.136,A -85,B 0,C 180,E1 -18968.968,E2 -18968.968} C_VEL
LIN {X 0,Y 257.678,Z 493.83,A -85,B 0,C 180,E1 -18970.895,E2 -18970.895} C_VEL
LIN {X 0,Y 255.593,Z 502.324,A -85,B 0,C 180,E1 -18973.219,E2 -18973.219} C_VEL
LIN {X 0,Y 253.781,Z 509.526,A -85,B 0,C 180,E1 -18975.759,E2 -18975.759} C_VEL
LIN {X 0,Y 252.62,Z 514.438,A -85,B 0,C 180,E1 -18977.956,E2 -18977.956} C_VEL
LIN {X 0,Y 251.377,Z 518.678,A -85,B 0,C 180,E1 -18980.343,E2 -18980.343} C_VEL
LIN {X 0,Y 250.748,Z 520.913,A -85,B 0,C 180,E1 -18981.944,E2 -18981.944} C_VEL
LIN {X 0,Y 250.215,Z 522.733,A -85,B 0,C 180,E1 -18983.549,E2 -18983.549} C_VEL
LIN {X 0,Y 249.791,Z 524.104,A -85,B 0,C 180,E1 -18985.158,E2 -18985.158} C_VEL
LIN {X 0,Y 249.645,Z 525.628,A -85,B 0,C 180,E1 -18988.387,E2 -18988.387} C_VEL
LIN {X 0,Y 249.616,Z 525.85,A -85,B 0,C 180,E1 -18990,E2 -18990} C_VEL
LIN {X 0,Y 249.644,Z 525.664,A -85,B 0,C 180,E1 -18991.613,E2 -18991.613} C_VEL
LIN {X 0,Y 249.782,Z 524.186,A -85,B 0,C 180,E1 -18994.842,E2 -18994.842} C_VEL
LIN {X 0,Y 250.2,Z 522.853,A -85,B 0,C 180,E1 -18996.451,E2 -18996.451} C_VEL
LIN {X 0,Y 251.098,Z 520.029,A -85,B 0,C 180,E1 -18998.855,E2 -18998.855} C_VEL
LIN {X 0,Y 252.212,Z 516.209,A -85,B 0,C 180,E1 -19001.248,E2 -19001.248} C_VEL
LIN {X 0,Y 253.586,Z 510.28,A -85,B 0,C 180,E1 -19004.067,E2 -19004.067} C_VEL
LIN {X 0,Y 255.586,Z 502.695,A -85,B 0,C 180,E1 -19006.782,E2 -19006.782} C_VEL
LIN {X 0,Y 257.609,Z 494.325,A -85,B 0,C 180,E1 -19009.11,E2 -19009.11} C_VEL
LIN {X 0,Y 259.347,Z 485.736,A -85,B 0,C 180,E1 -19011.042,E2 -19011.042} C_VEL
LIN {X 0,Y 261.301,Z 475.662,A -85,B 0,C 180,E1 -19012.855,E2 -19012.855} C_VEL
LIN {X 0,Y 258.997,Z 466.288,A -85,B 0,C 180,E1 -19014.693,E2 -19014.693} C_VEL
LIN {X 0,Y 255.544,Z 456.058,A -85,B 0,C 180,E1 -19016.513,E2 -19016.513} C_VEL
LIN {X 0,Y 251.329,Z 445.775,A -85,B 0,C 180,E1 -19018.169,E2 -19018.169} C_VEL
LIN {X 0,Y 249.208,Z 441.098,A -85,B 0,C 180,E1 -19018.872,E2 -19018.872} C_VEL
LIN {X 0,Y 249.073,Z 440.445,A -85,B 0,C 180,E1 -19018.988,E2 -19018.988} C_VEL
LIN {X 0,Y 249.038,Z 440.458,A -85,B 0,C 180,E1 -19022.425,E2 -19022.425} C_VEL
LIN {X 0,Y 249.078,Z 440.458,A -85,B 0,C 180,E1 -19026.337,E2 -19026.337} C_VEL
LIN {X 0,Y 249.1,Z 440.456,A -85,B 0,C 180,E1 -19030.46,E2 -19030.46} C_VEL
LIN {X 0,Y 249.076,Z 440.46,A -85,B 0,C 180,E1 -19032.809,E2 -19032.809} C_VEL
LIN {X 0,Y 249.026,Z 440.465,A -85,B 0,C 180,E1 -19037.365,E2 -19037.365} C_VEL
LIN {X 0,Y 249.027,Z 440.464,A -85,B 0,C 180,E1 -19041.619,E2 -19041.619} C_VEL
LIN {X 0,Y 249.045,Z 440.462,A -85,B 0,C 180,E1 -19045.639,E2 -19045.639} C_VEL
LIN {X 0,Y 249.049,Z 440.462,A -85,B 0,C 180,E1 -19049.473,E2 -19049.473} C_VEL
LIN {X 0,Y 249.073,Z 440.458,A -85,B 0,C 180,E1 -19053.162,E2 -19053.162} C_VEL
LIN {X 0,Y 249.082,Z 440.455,A -85,B 0,C 180,E1 -19056.733,E2 -19056.733} C_VEL
LIN {X 0,Y 249.113,Z 440.454,A -85,B 0,C 180,E1 -19060.212,E2 -19060.212} C_VEL
LIN {X 0,Y 249.244,Z 440.433,A -85,B 0,C 180,E1 -19063.622,E2 -19063.622} C_VEL
LIN {X 0,Y 249.247,Z 440.434,A -85,B 0,C 180,E1 -19068.616,E2 -19068.616} C_VEL
LIN {X 0,Y 249.448,Z 440.412,A -85,B 0,C 180,E1 -19071.902,E2 -19071.902} C_VEL
LIN {X 0,Y 249.297,Z 440.421,A -85,B 0,C 180,E1 -19075.148,E2 -19075.148} C_VEL
LIN {X 0,Y 249.679,Z 440.385,A -85,B 0,C 180,E1 -19078.387,E2 -19078.387} C_VEL
LIN {X 0,Y 249.679,Z 440.375,A -85,B 0,C 180,E1 -19081.613,E2 -19081.613} C_VEL
LIN {X 0,Y 249.45,Z 440.409,A -85,B 0,C 180,E1 -19086.471,E2 -19086.471} C_VEL
LIN {X 0,Y 249.345,Z 440.424,A -85,B 0,C 180,E1 -19089.736,E2 -19089.736} C_VEL
LIN {X 0,Y 249.208,Z 440.443,A -85,B 0,C 180,E1 -19094.703,E2 -19094.703} C_VEL
LIN {X 0,Y 249.141,Z 440.45,A -85,B 0,C 180,E1 -19098.077,E2 -19098.077} C_VEL
LIN {X 0,Y 249.086,Z 440.458,A -85,B 0,C 180,E1 -19101.518,E2 -19101.518} C_VEL
LIN {X 0,Y 249.119,Z 440.454,A -85,B 0,C 180,E1 -19105.476,E2 -19105.476} C_VEL
LIN {X 0,Y 249.075,Z 440.458,A -85,B 0,C 180,E1 -19108.989,E2 -19108.989} C_VEL
LIN {X 0,Y 249.037,Z 440.464,A -85,B 0,C 180,E1 -19112.425,E2 -19112.425} C_VEL
LIN {X 0,Y 249.098,Z 440.579,A -85,B 0,C 180,E1 -19115.29,E2 -19115.29} C_VEL
LIN {X 0,Y 250.27,Z 446.238,A -85,B 0,C 180,E1 -19119.186,E2 -19119.186} C_VEL
LIN {X 0,Y 250.792,Z 448.885,A -85,B 0,C 180,E1 -19120.899,E2 -19120.899} C_VEL
LIN {X 0,Y 250.484,Z 451.044,A -85,B 0,C 180,E1 -19122.153,E2 -19122.153} C_VEL
LIN {X 0,Y 248.367,Z 454.963,A -85,B 0,C 180,E1 -19124.186,E2 -19124.186} C_VEL
LIN {X 0,Y 246.566,Z 458.182,A -85,B 0,C 180,E1 -19125.829,E2 -19125.829} C_VEL
LIN {X 0,Y 245.959,Z 460.518,A -85,B 0,C 180,E1 -19127.099,E2 -19127.099} C_VEL
LIN {X 0,Y 246.004,Z 461.263,A -85,B 0,C 180,E1 -19127.528,E2 -19127.528} C_VEL
LIN {X 0,Y 246.798,Z 465.987,A -85,B 0,C 180,E1 -19130.253,E2 -19130.253} C_VEL
LIN {X 0,Y 246.28,Z 469.564,A -85,B 0,C 180,E1 -19132.154,E2 -19132.154} C_VEL
LIN {X 0,Y 244.409,Z 477.911,A -85,B 0,C 180,E1 -19136.502,E2 -19136.502} C_VEL
LIN {X 0,Y 243.414,Z 483.374,A -85,B 0,C 180,E1 -19139.288,E2 -19139.288} C_VEL
LIN {X 0,Y 245.995,Z 497.315,A -85,B 0,C 180,E1 -19140.347,E2 -19140.347} C_VEL
LIN {X 0,Y 247.492,Z 509.096,A -85,B 0,C 180,E1 -19141.448,E2 -19141.448} C_VEL
LIN {X 0,Y 248.268,Z 521.681,A -85,B 0,C 180,E1 -19142.855,E2 -19142.855} C_VEL
LIN {X 0,Y 248.331,Z 533.34,A -85,B 0,C 180,E1 -19144.432,E2 -19144.432} C_VEL
LIN {X 0,Y 247.786,Z 544.302,A -85,B 0,C 180,E1 -19146.205,E2 -19146.205} C_VEL
LIN {X 0,Y 246.793,Z 554.879,A -85,B 0,C 180,E1 -19148.272,E2 -19148.272} C_VEL
LIN {X 0,Y 245.095,Z 563.55,A -85,B 0,C 180,E1 -19150.31,E2 -19150.31} C_VEL
LIN {X 0,Y 243.425,Z 570.965,A -85,B 0,C 180,E1 -19152.429,E2 -19152.429} C_VEL
LIN {X 0,Y 242.049,Z 577.842,A -85,B 0,C 180,E1 -19154.852,E2 -19154.852} C_VEL
LIN {X 0,Y 241.203,Z 583.59,A -85,B 0,C 180,E1 -19157.377,E2 -19157.377} C_VEL
LIN {X 0,Y 240.816,Z 588.147,A -85,B 0,C 180,E1 -19159.915,E2 -19159.915} C_VEL
LIN {X 0,Y 240.895,Z 591.936,A -85,B 0,C 180,E1 -19162.72,E2 -19162.72} C_VEL
LIN {X 0,Y 241.214,Z 594.117,A -85,B 0,C 180,E1 -19164.986,E2 -19164.986} C_VEL
LIN {X 0,Y 241.47,Z 595.215,A -85,B 0,C 180,E1 -19166.663,E2 -19166.663} C_VEL
LIN {X 0,Y 242.15,Z 596.183,A -85,B 0,C 180,E1 -19170,E2 -19170} C_VEL
LIN {X 0,Y 241.469,Z 595.2,A -85,B 0,C 180,E1 -19173.337,E2 -19173.337} C_VEL
LIN {X 0,Y 241.214,Z 594.098,A -85,B 0,C 180,E1 -19175.015,E2 -19175.015} C_VEL
LIN {X 0,Y 240.898,Z 591.898,A -85,B 0,C 180,E1 -19177.286,E2 -19177.286} C_VEL
LIN {X 0,Y 240.816,Z 588.097,A -85,B 0,C 180,E1 -19180.085,E2 -19180.085} C_VEL
LIN {X 0,Y 241.202,Z 583.522,A -85,B 0,C 180,E1 -19182.623,E2 -19182.623} C_VEL
LIN {X 0,Y 242.037,Z 577.757,A -85,B 0,C 180,E1 -19185.149,E2 -19185.149} C_VEL
LIN {X 0,Y 243.084,Z 571.883,A -85,B 0,C 180,E1 -19187.241,E2 -19187.241} C_VEL
LIN {X 0,Y 244.763,Z 564.947,A -85,B 0,C 180,E1 -19189.281,E2 -19189.281} C_VEL
LIN {X 0,Y 246.511,Z 556.575,A -85,B 0,C 180,E1 -19191.316,E2 -19191.316} C_VEL
LIN {X 0,Y 247.594,Z 546.253,A -85,B 0,C 180,E1 -19193.415,E2 -19193.415} C_VEL
LIN {X 0,Y 248.219,Z 536.039,A -85,B 0,C 180,E1 -19195.132,E2 -19195.132} C_VEL
LIN {X 0,Y 248.29,Z 524.908,A -85,B 0,C 180,E1 -19196.702,E2 -19196.702} C_VEL
LIN {X 0,Y 247.716,Z 512.039,A -85,B 0,C 180,E1 -19198.203,E2 -19198.203} C_VEL
LIN {X 0,Y 246.149,Z 498.628,A -85,B 0,C 180,E1 -19199.506,E2 -19199.506} C_VEL
LIN {X 0,Y 243.587,Z 485.171,A -85,B 0,C 180,E1 -19200.572,E2 -19200.572} C_VEL
LIN {X 0,Y 243.39,Z 483.148,A -85,B 0,C 180,E1 -19200.747,E2 -19200.747} C_VEL
LIN {X 0,Y 245.06,Z 474.919,A -85,B 0,C 180,E1 -19205,E2 -19205} C_VEL
LIN {X 0,Y 246.659,Z 467.573,A -85,B 0,C 180,E1 -19208.818,E2 -19208.818} C_VEL
LIN {X 0,Y 246.677,Z 464.918,A -85,B 0,C 180,E1 -19210.269,E2 -19210.269} C_VEL
LIN {X 0,Y 245.411,Z 458.166,A -85,B 0,C 180,E1 -19214.279,E2 -19214.279} C_VEL
LIN {X 0,Y 244.061,Z 451.369,A -85,B 0,C 180,E1 -19218.524,E2 -19218.524} C_VEL
LIN {X 0,Y 242.901,Z 445.416,A -85,B 0,C 180,E1 -19222.583,E2 -19222.583} C_VEL
LIN {X 0,Y 242.037,Z 441.337,A -85,B 0,C 180,E1 -19225.639,E2 -19225.639} C_VEL
LIN {X 0,Y 242.016,Z 441.342,A -85,B 0,C 180,E1 -19230.597,E2 -19230.597} C_VEL
LIN {X 0,Y 242.07,Z 441.331,A -85,B 0,C 180,E1 -19234.183,E2 -19234.183} C_VEL
LIN {X 0,Y 242.029,Z 441.333,A -85,B 0,C 180,E1 -19238.313,E2 -19238.313} C_VEL
LIN {X 0,Y 242.166,Z 441.32,A -85,B 0,C 180,E1 -19243.278,E2 -19243.278} C_VEL
LIN {X 0,Y 242.184,Z 441.32,A -85,B 0,C 180,E1 -19248.28,E2 -19248.28} C_VEL
LIN {X 0,Y 242.397,Z 441.294,A -85,B 0,C 180,E1 -19251.665,E2 -19251.665} C_VEL
LIN {X 0,Y 242.261,Z 441.309,A -85,B 0,C 180,E1 -19255.007,E2 -19255.007} C_VEL
LIN {X 0,Y 242.641,Z 441.261,A -85,B 0,C 180,E1 -19258.34,E2 -19258.34} C_VEL
LIN {X 0,Y 242.64,Z 441.263,A -85,B 0,C 180,E1 -19261.66,E2 -19261.66} C_VEL
LIN {X 0,Y 242.42,Z 441.285,A -85,B 0,C 180,E1 -19266.669,E2 -19266.669} C_VEL
LIN {X 0,Y 242.27,Z 441.304,A -85,B 0,C 180,E1 -19270.024,E2 -19270.024} C_VEL
LIN {X 0,Y 242.17,Z 441.281,A -85,B 0,C 180,E1 -19275.141,E2 -19275.141} C_VEL
LIN {X 0,Y 242.076,Z 441.315,A -85,B 0,C 180,E1 -19278.624,E2 -19278.624} C_VEL
LIN {X 0,Y 242.016,Z 441.335,A -85,B 0,C 180,E1 -19282.18,E2 -19282.18} C_VEL
LIN {X 0,Y 242.069,Z 441.311,A -85,B 0,C 180,E1 -19285.838,E2 -19285.838} C_VEL
LIN {X 0,Y 242.01,Z 441.318,A -85,B 0,C 180,E1 -19289.583,E2 -19289.583} C_VEL
LIN {X 0,Y 241.983,Z 441.341,A -85,B 0,C 180,E1 -19293.492,E2 -19293.492} C_VEL
LIN {X 0,Y 241.989,Z 441.342,A -85,B 0,C 180,E1 -19297.582,E2 -19297.582} C_VEL
LIN {X 0,Y 241.946,Z 441.346,A -85,B 0,C 180,E1 -19301.921,E2 -19301.921} C_VEL
LIN {X 0,Y 242.004,Z 441.339,A -85,B 0,C 180,E1 -19306.554,E2 -19306.554} C_VEL
LIN {X 0,Y 242.013,Z 441.334,A -85,B 0,C 180,E1 -19310.292,E2 -19310.292} C_VEL
LIN {X 0,Y 242.039,Z 441.33,A -85,B 0,C 180,E1 -19314.498,E2 -19314.498} C_VEL
LIN {X 0,Y 242.019,Z 441.337,A -85,B 0,C 180,E1 -19319.458,E2 -19319.458} C_VEL
LIN {X 0,Y 242.017,Z 441.337,A -85,B 0,C 180,E1 -19320.243,E2 -19320.243} C_VEL
LIN {X 0,Y 242.564,Z 443.286,A -85,B 0,C 180,E1 -19320.491,E2 -19320.491} C_VEL
LIN {X 0,Y 247.472,Z 453.943,A -85,B 0,C 180,E1 -19322.282,E2 -19322.282} C_VEL
LIN {X 0,Y 251.188,Z 464.405,A -85,B 0,C 180,E1 -19324.157,E2 -19324.157} C_VEL
LIN {X 0,Y 253.87,Z 473.692,A -85,B 0,C 180,E1 -19326.002,E2 -19326.002} C_VEL
LIN {X 0,Y 254.638,Z 477.025,A -85,B 0,C 180,E1 -19326.708,E2 -19326.708} C_VEL
LIN {X 0,Y 252.929,Z 486.143,A -85,B 0,C 180,E1 -19328.397,E2 -19328.397} C_VEL
LIN {X 0,Y 251.049,Z 494.838,A -85,B 0,C 180,E1 -19330.37,E2 -19330.37} C_VEL
LIN {X 0,Y 248.873,Z 503.332,A -85,B 0,C 180,E1 -19332.752,E2 -19332.752} C_VEL
LIN {X 0,Y 246.977,Z 510.528,A -85,B 0,C 180,E1 -19335.356,E2 -19335.356} C_VEL
LIN {X 0,Y 245.751,Z 515.444,A -85,B 0,C 180,E1 -19337.614,E2 -19337.614} C_VEL
LIN {X 0,Y 244.452,Z 519.684,A -85,B 0,C 180,E1 -19340.067,E2 -19340.067} C_VEL
LIN {X 0,Y 243.792,Z 521.919,A -85,B 0,C 180,E1 -19341.712,E2 -19341.712} C_VEL
LIN {X 0,Y 243.233,Z 523.739,A -85,B 0,C 180,E1 -19343.363,E2 -19343.363} C_VEL
LIN {X 0,Y 242.789,Z 525.109,A -85,B 0,C 180,E1 -19345.018,E2 -19345.018} C_VEL
LIN {X 0,Y 242.621,Z 526.633,A -85,B 0,C 180,E1 -19348.34,E2 -19348.34} C_VEL
LIN {X 0,Y 242.59,Z 526.854,A -85,B 0,C 180,E1 -19350,E2 -19350} C_VEL
LIN {X 0,Y 242.62,Z 526.668,A -85,B 0,C 180,E1 -19351.66,E2 -19351.66} C_VEL
LIN {X 0,Y 242.779,Z 525.19,A -85,B 0,C 180,E1 -19354.982,E2 -19354.982} C_VEL
LIN {X 0,Y 243.217,Z 523.857,A -85,B 0,C 180,E1 -19356.637,E2 -19356.637} C_VEL
LIN {X 0,Y 244.157,Z 521.034,A -85,B 0,C 180,E1 -19359.109,E2 -19359.109} C_VEL
LIN {X 0,Y 245.323,Z 517.213,A -85,B 0,C 180,E1 -19361.568,E2 -19361.568} C_VEL
LIN {X 0,Y 246.773,Z 511.288,A -85,B 0,C 180,E1 -19364.463,E2 -19364.463} C_VEL
LIN {X 0,Y 248.865,Z 503.698,A -85,B 0,C 180,E1 -19367.249,E2 -19367.249} C_VEL
LIN {X 0,Y 250.979,Z 495.327,A -85,B 0,C 180,E1 -19369.635,E2 -19369.635} C_VEL
LIN {X 0,Y 252.804,Z 486.737,A -85,B 0,C 180,E1 -19371.614,E2 -19371.614} C_VEL
LIN {X 0,Y 254.67,Z 477.298,A -85,B 0,C 180,E1 -19373.368,E2 -19373.368} C_VEL
LIN {X 0,Y 252.451,Z 468.28,A -85,B 0,C 180,E1 -19375.222,E2 -19375.222} C_VEL
LIN {X 0,Y 248.917,Z 457.728,A -85,B 0,C 180,E1 -19377.202,E2 -19377.202} C_VEL
LIN {X 0,Y 244.836,Z 447.784,A -85,B 0,C 180,E1 -19378.897,E2 -19378.897} C_VEL
LIN {X 0,Y 242.151,Z 442.169,A -85,B 0,C 180,E1 -19379.803,E2 -19379.803} C_VEL
LIN {X 0,Y 241.999,Z 441.333,A -85,B 0,C 180,E1 -19379.943,E2 -19379.943} C_VEL
LIN {X 0,Y 241.993,Z 441.34,A -85,B 0,C 180,E1 -19383.491,E2 -19383.491} C_VEL
LIN {X 0,Y 242.022,Z 441.338,A -85,B 0,C 180,E1 -19387.576,E2 -19387.576} C_VEL
LIN {X 0,Y 242.032,Z 441.335,A -85,B 0,C 180,E1 -19391.902,E2 -19391.902} C_VEL
LIN {X 0,Y 241.946,Z 441.348,A -85,B 0,C 180,E1 -19396.569,E2 -19396.569} C_VEL
LIN {X 0,Y 241.969,Z 441.344,A -85,B 0,C 180,E1 -19400.283,E2 -19400.283} C_VEL
LIN {X 0,Y 241.982,Z 441.342,A -85,B 0,C 180,E1 -19404.488,E2 -19404.488} C_VEL
LIN {X 0,Y 241.974,Z 441.34,A -85,B 0,C 180,E1 -19408.48,E2 -19408.48} C_VEL
LIN {X 0,Y 242.004,Z 441.336,A -85,B 0,C 180,E1 -19412.312,E2 -19412.312} C_VEL
LIN {X 0,Y 242.059,Z 441.332,A -85,B 0,C 180,E1 -19416.016,E2 -19416.016} C_VEL
LIN {X 0,Y 242.04,Z 441.334,A -85,B 0,C 180,E1 -19419.608,E2 -19419.608} C_VEL
LIN {X 0,Y 242.165,Z 441.316,A -85,B 0,C 180,E1 -19423.278,E2 -19423.278} C_VEL
LIN {X 0,Y 242.184,Z 441.312,A -85,B 0,C 180,E1 -19428.28,E2 -19428.28} C_VEL
LIN {X 0,Y 242.396,Z 441.29,A -85,B 0,C 180,E1 -19431.664,E2 -19431.664} C_VEL
LIN {X 0,Y 242.258,Z 441.297,A -85,B 0,C 180,E1 -19435.007,E2 -19435.007} C_VEL
LIN {X 0,Y 242.639,Z 441.262,A -85,B 0,C 180,E1 -19438.34,E2 -19438.34} C_VEL
LIN {X 0,Y 242.639,Z 441.251,A -85,B 0,C 180,E1 -19441.66,E2 -19441.66} C_VEL
LIN {X 0,Y 242.42,Z 441.283,A -85,B 0,C 180,E1 -19446.659,E2 -19446.659} C_VEL
LIN {X 0,Y 242.269,Z 441.306,A -85,B 0,C 180,E1 -19450.024,E2 -19450.024} C_VEL
LIN {X 0,Y 242.169,Z 441.318,A -85,B 0,C 180,E1 -19455.141,E2 -19455.141} C_VEL
LIN {X 0,Y 242.075,Z 441.332,A -85,B 0,C 180,E1 -19458.624,E2 -19458.624} C_VEL
LIN {X 0,Y 242.008,Z 441.342,A -85,B 0,C 180,E1 -19462.18,E2 -19462.18} C_VEL
LIN {X 0,Y 242.068,Z 441.334,A -85,B 0,C 180,E1 -19465.838,E2 -19465.838} C_VEL
LIN {X 0,Y 242.008,Z 441.337,A -85,B 0,C 180,E1 -19469.583,E2 -19469.583} C_VEL
LIN {X 0,Y 242.055,Z 441.472,A -85,B 0,C 180,E1 -19474.484,E2 -19474.484} C_VEL
LIN {X 0,Y 243.301,Z 447.409,A -85,B 0,C 180,E1 -19478.746,E2 -19478.746} C_VEL
LIN {X 0,Y 244.709,Z 454.779,A -85,B 0,C 180,E1 -19483.573,E2 -19483.573} C_VEL
LIN {X 0,Y 246.004,Z 461.263,A -85,B 0,C 180,E1 -19487.528,E2 -19487.528} C_VEL
LIN {X 0,Y 245.59,Z 463.583,A -85,B 0,C 180,E1 -19488.789,E2 -19488.789} C_VEL
LIN {X 0,Y 244.077,Z 466.056,A -85,B 0,C 180,E1 -19490.007,E2 -19490.007} C_VEL
LIN {X 0,Y 238.926,Z 472.779,A -85,B 0,C 180,E1 -19493.273,E2 -19493.273} C_VEL
LIN {X 0,Y 238.301,Z 474.432,A -85,B 0,C 180,E1 -19494.145,E2 -19494.145} C_VEL
LIN {X 0,Y 236.623,Z 482.142,A -85,B 0,C 180,E1 -19498.292,E2 -19498.292} C_VEL
LIN {X 0,Y 239.368,Z 497.041,A -85,B 0,C 180,E1 -19499.492,E2 -19499.492} C_VEL
LIN {X 0,Y 240.808,Z 508.145,A -85,B 0,C 180,E1 -19500.591,E2 -19500.591} C_VEL
LIN {X 0,Y 241.572,Z 520.912,A -85,B 0,C 180,E1 -19502.077,E2 -19502.077} C_VEL
LIN {X 0,Y 241.639,Z 532.28,A -85,B 0,C 180,E1 -19503.67,E2 -19503.67} C_VEL
LIN {X 0,Y 241.051,Z 543.581,A -85,B 0,C 180,E1 -19505.559,E2 -19505.559} C_VEL
LIN {X 0,Y 240.038,Z 553.84,A -85,B 0,C 180,E1 -19507.628,E2 -19507.628} C_VEL
LIN {X 0,Y 238.758,Z 560.913,A -85,B 0,C 180,E1 -19509.315,E2 -19509.315} C_VEL
LIN {X 0,Y 236.771,Z 569.553,A -85,B 0,C 180,E1 -19511.777,E2 -19511.777} C_VEL
LIN {X 0,Y 235.558,Z 574.604,A -85,B 0,C 180,E1 -19513.535,E2 -19513.535} C_VEL
LIN {X 0,Y 234.483,Z 580.798,A -85,B 0,C 180,E1 -19516.127,E2 -19516.127} C_VEL
LIN {X 0,Y 233.835,Z 585.734,A -85,B 0,C 180,E1 -19518.734,E2 -19518.734} C_VEL
LIN {X 0,Y 233.749,Z 589.57,A -85,B 0,C 180,E1 -19521.354,E2 -19521.354} C_VEL
LIN {X 0,Y 233.877,Z 591.574,A -85,B 0,C 180,E1 -19523.096,E2 -19523.096} C_VEL
LIN {X 0,Y 234.125,Z 593.1,A -85,B 0,C 180,E1 -19524.833,E2 -19524.833} C_VEL
LIN {X 0,Y 234.409,Z 594.203,A -85,B 0,C 180,E1 -19526.562,E2 -19526.562} C_VEL
LIN {X 0,Y 235.114,Z 595.177,A -85,B 0,C 180,E1 -19530,E2 -19530} C_VEL
LIN {X 0,Y 234.408,Z 594.188,A -85,B 0,C 180,E1 -19533.438,E2 -19533.438} C_VEL
LIN {X 0,Y 234.125,Z 593.08,A -85,B 0,C 180,E1 -19535.167,E2 -19535.167} C_VEL
LIN {X 0,Y 233.826,Z 591.093,A -85,B 0,C 180,E1 -19537.313,E2 -19537.313} C_VEL
LIN {X 0,Y 233.744,Z 587.068,A -85,B 0,C 180,E1 -19540.393,E2 -19540.393} C_VEL
LIN {X 0,Y 234.208,Z 582.495,A -85,B 0,C 180,E1 -19543.006,E2 -19543.006} C_VEL
LIN {X 0,Y 235.116,Z 576.728,A -85,B 0,C 180,E1 -19545.606,E2 -19545.606} C_VEL
LIN {X 0,Y 236.309,Z 570.835,A -85,B 0,C 180,E1 -19547.762,E2 -19547.762} C_VEL
LIN {X 0,Y 238.005,Z 563.919,A -85,B 0,C 180,E1 -19549.852,E2 -19549.852} C_VEL
LIN {X 0,Y 239.77,Z 555.535,A -85,B 0,C 180,E1 -19551.946,E2 -19551.946} C_VEL
LIN {X 0,Y 240.88,Z 545.2,A -85,B 0,C 180,E1 -19554.109,E2 -19554.109} C_VEL
LIN {X 0,Y 241.524,Z 534.974,A -85,B 0,C 180,E1 -19555.88,E2 -19555.88} C_VEL
LIN {X 0,Y 241.609,Z 523.829,A -85,B 0,C 180,E1 -19557.502,E2 -19557.502} C_VEL
LIN {X 0,Y 241.053,Z 511.546,A -85,B 0,C 180,E1 -19558.995,E2 -19558.995} C_VEL
LIN {X 0,Y 239.565,Z 498.24,A -85,B 0,C 180,E1 -19560.347,E2 -19560.347} C_VEL
LIN {X 0,Y 236.927,Z 484.505,A -85,B 0,C 180,E1 -19561.51,E2 -19561.51} C_VEL
LIN {X 0,Y 236.62,Z 482.127,A -85,B 0,C 180,E1 -19561.671,E2 -19561.671} C_VEL
LIN {X 0,Y 238.396,Z 473.796,A -85,B 0,C 180,E1 -19566.13,E2 -19566.13} C_VEL
LIN {X 0,Y 239.67,Z 468.332,A -85,B 0,C 180,E1 -19569.084,E2 -19569.084} C_VEL
LIN {X 0,Y 239.705,Z 466.122,A -85,B 0,C 180,E1 -19570.332,E2 -19570.332} C_VEL
LIN {X 0,Y 238.622,Z 460.388,A -85,B 0,C 180,E1 -19573.814,E2 -19573.814} C_VEL
LIN {X 0,Y 237.166,Z 453.102,A -85,B 0,C 180,E1 -19578.508,E2 -19578.508} C_VEL
LIN {X 0,Y 236.082,Z 447.515,A -85,B 0,C 180,E1 -19582.391,E2 -19582.391} C_VEL
LIN {X 0,Y 234.97,Z 442.214,A -85,B 0,C 180,E1 -19586.522,E2 -19586.522} C_VEL
LIN {X 0,Y 234.938,Z 442.221,A -85,B 0,C 180,E1 -19591.404,E2 -19591.404} C_VEL
LIN {X 0,Y 234.98,Z 442.213,A -85,B 0,C 180,E1 -19595.246,E2 -19595.246} C_VEL
LIN {X 0,Y 235.001,Z 442.21,A -85,B 0,C 180,E1 -19598.969,E2 -19598.969} C_VEL
LIN {X 0,Y 235.099,Z 442.2,A -85,B 0,C 180,E1 -19603.059,E2 -19603.059} C_VEL
LIN {X 0,Y 235.118,Z 442.2,A -85,B 0,C 180,E1 -19607.922,E2 -19607.922} C_VEL
LIN {X 0,Y 235.329,Z 442.173,A -85,B 0,C 180,E1 -19611.412,E2 -19611.412} C_VEL
LIN {X 0,Y 235.371,Z 442.168,A -85,B 0,C 180,E1 -19613.14,E2 -19613.14} C_VEL
LIN {X 0,Y 235.6,Z 442.138,A -85,B 0,C 180,E1 -19618.291,E2 -19618.291} C_VEL
LIN {X 0,Y 235.599,Z 442.14,A -85,B 0,C 180,E1 -19621.709,E2 -19621.709} C_VEL
LIN {X 0,Y 235.371,Z 442.164,A -85,B 0,C 180,E1 -19626.86,E2 -19626.86} C_VEL
LIN {X 0,Y 235.217,Z 442.182,A -85,B 0,C 180,E1 -19630.328,E2 -19630.328} C_VEL
LIN {X 0,Y 235.117,Z 442.156,A -85,B 0,C 180,E1 -19635.606,E2 -19635.606} C_VEL
LIN {X 0,Y 235.012,Z 442.196,A -85,B 0,C 180,E1 -19639.205,E2 -19639.205} C_VEL
LIN {X 0,Y 234.964,Z 442.214,A -85,B 0,C 180,E1 -19642.883,E2 -19642.883} C_VEL
LIN {X 0,Y 234.97,Z 442.186,A -85,B 0,C 180,E1 -19646.657,E2 -19646.657} C_VEL
LIN {X 0,Y 234.925,Z 442.21,A -85,B 0,C 180,E1 -19650.569,E2 -19650.569} C_VEL
LIN {X 0,Y 234.929,Z 442.218,A -85,B 0,C 180,E1 -19654.638,E2 -19654.638} C_VEL
LIN {X 0,Y 234.944,Z 442.217,A -85,B 0,C 180,E1 -19658.944,E2 -19658.944} C_VEL
LIN {X 0,Y 234.925,Z 442.217,A -85,B 0,C 180,E1 -19663.478,E2 -19663.478} C_VEL
LIN {X 0,Y 234.977,Z 442.214,A -85,B 0,C 180,E1 -19666.534,E2 -19666.534} C_VEL
LIN {X 0,Y 234.973,Z 442.21,A -85,B 0,C 180,E1 -19671.089,E2 -19671.089} C_VEL
LIN {X 0,Y 234.963,Z 442.211,A -85,B 0,C 180,E1 -19675.367,E2 -19675.367} C_VEL
LIN {X 0,Y 234.979,Z 442.212,A -85,B 0,C 180,E1 -19679.221,E2 -19679.221} C_VEL
LIN {X 0,Y 236.103,Z 445.224,A -85,B 0,C 180,E1 -19679.682,E2 -19679.682} C_VEL
LIN {X 0,Y 240.948,Z 455.846,A -85,B 0,C 180,E1 -19681.568,E2 -19681.568} C_VEL
LIN {X 0,Y 244.505,Z 465.934,A -85,B 0,C 180,E1 -19683.466,E2 -19683.466} C_VEL
LIN {X 0,Y 247.247,Z 475.472,A -85,B 0,C 180,E1 -19685.451,E2 -19685.451} C_VEL
LIN {X 0,Y 248.036,Z 479.519,A -85,B 0,C 180,E1 -19686.34,E2 -19686.34} C_VEL
LIN {X 0,Y 245.989,Z 489.065,A -85,B 0,C 180,E1 -19688.197,E2 -19688.197} C_VEL
LIN {X 0,Y 244.063,Z 497.418,A -85,B 0,C 180,E1 -19690.223,E2 -19690.223} C_VEL
LIN {X 0,Y 241.846,Z 505.542,A -85,B 0,C 180,E1 -19692.67,E2 -19692.67} C_VEL
LIN {X 0,Y 240.185,Z 511.532,A -85,B 0,C 180,E1 -19694.93,E2 -19694.93} C_VEL
LIN {X 0,Y 238.892,Z 516.451,A -85,B 0,C 180,E1 -19697.253,E2 -19697.253} C_VEL
LIN {X 0,Y 237.533,Z 520.69,A -85,B 0,C 180,E1 -19699.774,E2 -19699.774} C_VEL
LIN {X 0,Y 236.84,Z 522.925,A -85,B 0,C 180,E1 -19701.467,E2 -19701.467} C_VEL
LIN {X 0,Y 236.253,Z 524.745,A -85,B 0,C 180,E1 -19703.166,E2 -19703.166} C_VEL
LIN {X 0,Y 235.788,Z 526.115,A -85,B 0,C 180,E1 -19704.87,E2 -19704.87} C_VEL
LIN {X 0,Y 235.597,Z 527.638,A -85,B 0,C 180,E1 -19708.29,E2 -19708.29} C_VEL
LIN {X 0,Y 235.564,Z 527.859,A -85,B 0,C 180,E1 -19710,E2 -19710} C_VEL
LIN {X 0,Y 235.596,Z 527.673,A -85,B 0,C 180,E1 -19711.709,E2 -19711.709} C_VEL
LIN {X 0,Y 235.778,Z 526.195,A -85,B 0,C 180,E1 -19715.13,E2 -19715.13} C_VEL
LIN {X 0,Y 236.238,Z 524.862,A -85,B 0,C 180,E1 -19716.834,E2 -19716.834} C_VEL
LIN {X 0,Y 237.22,Z 522.038,A -85,B 0,C 180,E1 -19719.378,E2 -19719.378} C_VEL
LIN {X 0,Y 238.442,Z 518.217,A -85,B 0,C 180,E1 -19721.907,E2 -19721.907} C_VEL
LIN {X 0,Y 239.973,Z 512.295,A -85,B 0,C 180,E1 -19724.88,E2 -19724.88} C_VEL
LIN {X 0,Y 241.841,Z 505.901,A -85,B 0,C 180,E1 -19727.33,E2 -19727.33} C_VEL
LIN {X 0,Y 244.009,Z 497.86,A -85,B 0,C 180,E1 -19729.781,E2 -19729.781} C_VEL
LIN {X 0,Y 245.883,Z 489.633,A -85,B 0,C 180,E1 -19731.813,E2 -19731.813} C_VEL
LIN {X 0,Y 247.928,Z 480.316,A -85,B 0,C 180,E1 -19733.652,E2 -19733.652} C_VEL
LIN {X 0,Y 248.041,Z 478.934,A -85,B 0,C 180,E1 -19733.911,E2 -19733.911} C_VEL
LIN {X 0,Y 245.791,Z 469.952,A -85,B 0,C 180,E1 -19735.852,E2 -19735.852} C_VEL
LIN {X 0,Y 242.453,Z 459.744,A -85,B 0,C 180,E1 -19737.856,E2 -19737.856} C_VEL
LIN {X 0,Y 238.448,Z 450.179,A -85,B 0,C 180,E1 -19739.603,E2 -19739.603} C_VEL
LIN {X 0,Y 235.098,Z 442.908,A -85,B 0,C 180,E1 -19740.827,E2 -19740.827} C_VEL
LIN {X 0,Y 234.966,Z 442.215,A -85,B 0,C 180,E1 -19740.936,E2 -19740.936} C_VEL
LIN {X 0,Y 234.962,Z 442.213,A -85,B 0,C 180,E1 -19744.633,E2 -19744.633} C_VEL
LIN {X 0,Y 234.999,Z 442.213,A -85,B 0,C 180,E1 -19748.961,E2 -19748.961} C_VEL
LIN {X 0,Y 234.976,Z 442.215,A -85,B 0,C 180,E1 -19753.465,E2 -19753.465} C_VEL
LIN {X 0,Y 234.924,Z 442.222,A -85,B 0,C 180,E1 -19756.522,E2 -19756.522} C_VEL
LIN {X 0,Y 234.925,Z 442.224,A -85,B 0,C 180,E1 -19761.08,E2 -19761.08} C_VEL
LIN {X 0,Y 234.928,Z 442.222,A -85,B 0,C 180,E1 -19765.361,E2 -19765.361} C_VEL
LIN {X 0,Y 234.924,Z 442.222,A -85,B 0,C 180,E1 -19769.431,E2 -19769.431} C_VEL
LIN {X 0,Y 234.995,Z 442.21,A -85,B 0,C 180,E1 -19773.794,E2 -19773.794} C_VEL
LIN {X 0,Y 235.013,Z 442.21,A -85,B 0,C 180,E1 -19778.97,E2 -19778.97} C_VEL
LIN {X 0,Y 235.098,Z 442.195,A -85,B 0,C 180,E1 -19783.059,E2 -19783.059} C_VEL
LIN {X 0,Y 235.117,Z 442.193,A -85,B 0,C 180,E1 -19787.922,E2 -19787.922} C_VEL
LIN {X 0,Y 235.328,Z 442.17,A -85,B 0,C 180,E1 -19791.412,E2 -19791.412} C_VEL
LIN {X 0,Y 235.37,Z 442.16,A -85,B 0,C 180,E1 -19793.14,E2 -19793.14} C_VEL
LIN {X 0,Y 235.598,Z 442.138,A -85,B 0,C 180,E1 -19798.291,E2 -19798.291} C_VEL
LIN {X 0,Y 235.599,Z 442.127,A -85,B 0,C 180,E1 -19801.709,E2 -19801.709} C_VEL
LIN {X 0,Y 235.37,Z 442.16,A -85,B 0,C 180,E1 -19806.86,E2 -19806.86} C_VEL
LIN {X 0,Y 235.216,Z 442.187,A -85,B 0,C 180,E1 -19810.327,E2 -19810.327} C_VEL
LIN {X 0,Y 235.116,Z 442.198,A -85,B 0,C 180,E1 -19815.606,E2 -19815.606} C_VEL
LIN {X 0,Y 235.01,Z 442.211,A -85,B 0,C 180,E1 -19819.205,E2 -19819.205} C_VEL
LIN {X 0,Y 234.954,Z 442.218,A -85,B 0,C 180,E1 -19822.884,E2 -19822.884} C_VEL
LIN {X 0,Y 234.969,Z 442.217,A -85,B 0,C 180,E1 -19826.657,E2 -19826.657} C_VEL
LIN {X 0,Y 234.924,Z 442.223,A -85,B 0,C 180,E1 -19830.569,E2 -19830.569} C_VEL
LIN {X 0,Y 234.956,Z 442.296,A -85,B 0,C 180,E1 -19833.585,E2 -19833.585} C_VEL
LIN {X 0,Y 236.134,Z 447.626,A -85,B 0,C 180,E1 -19837.599,E2 -19837.599} C_VEL
LIN {X 0,Y 237.406,Z 454.402,A -85,B 0,C 180,E1 -19842.262,E2 -19842.262} C_VEL
LIN {X 0,Y 238.627,Z 460.519,A -85,B 0,C 180,E1 -19846.184,E2 -19846.184} C_VEL
LIN {X 0,Y 239.735,Z 466.552,A -85,B 0,C 180,E1 -19849.838,E2 -19849.838} C_VEL
LIN {X 0,Y 239.668,Z 468.455,A -85,B 0,C 180,E1 -19850.916,E2 -19850.916} C_VEL
LIN {X 0,Y 238.301,Z 474.432,A -85,B 0,C 180,E1 -19854.145,E2 -19854.145} C_VEL
LIN {X 0,Y 237.396,Z 477.355,A -85,B 0,C 180,E1 -19855.321,E2 -19855.321} C_VEL
LIN {X 0,Y 235.982,Z 481.175,A -85,B 0,C 180,E1 -19856.324,E2 -19856.324} C_VEL
LIN {X 0,Y 234.038,Z 487.236,A -85,B 0,C 180,E1 -19857.43,E2 -19857.43} C_VEL
LIN {X 0,Y 233.051,Z 492.321,A -85,B 0,C 180,E1 -19858.119,E2 -19858.119} C_VEL
LIN {X 0,Y 232.982,Z 497.697,A -85,B 0,C 180,E1 -19858.696,E2 -19858.696} C_VEL
LIN {X 0,Y 234.375,Z 509.564,A -85,B 0,C 180,E1 -19859.955,E2 -19859.955} C_VEL
LIN {X 0,Y 234.962,Z 521.257,A -85,B 0,C 180,E1 -19861.407,E2 -19861.407} C_VEL
LIN {X 0,Y 234.932,Z 532.7,A -85,B 0,C 180,E1 -19863.098,E2 -19863.098} C_VEL
LIN {X 0,Y 234.192,Z 544.35,A -85,B 0,C 180,E1 -19865.157,E2 -19865.157} C_VEL
LIN {X 0,Y 233.04,Z 554.656,A -85,B 0,C 180,E1 -19867.387,E2 -19867.387} C_VEL
LIN {X 0,Y 231.683,Z 561.509,A -85,B 0,C 180,E1 -19869.119,E2 -19869.119} C_VEL
LIN {X 0,Y 229.528,Z 570.218,A -85,B 0,C 180,E1 -19871.798,E2 -19871.798} C_VEL
LIN {X 0,Y 228.239,Z 575.794,A -85,B 0,C 180,E1 -19873.911,E2 -19873.911} C_VEL
LIN {X 0,Y 227.237,Z 581.542,A -85,B 0,C 180,E1 -19876.588,E2 -19876.588} C_VEL
LIN {X 0,Y 226.704,Z 586.097,A -85,B 0,C 180,E1 -19879.28,E2 -19879.28} C_VEL
LIN {X 0,Y 226.777,Z 590.28,A -85,B 0,C 180,E1 -19882.617,E2 -19882.617} C_VEL
LIN {X 0,Y 227.042,Z 592.083,A -85,B 0,C 180,E1 -19884.672,E2 -19884.672} C_VEL
LIN {X 0,Y 227.346,Z 593.191,A -85,B 0,C 180,E1 -19886.455,E2 -19886.455} C_VEL
LIN {X 0,Y 228.076,Z 594.17,A -85,B 0,C 180,E1 -19890,E2 -19890} C_VEL
LIN {X 0,Y 227.345,Z 593.176,A -85,B 0,C 180,E1 -19893.545,E2 -19893.545} C_VEL
LIN {X 0,Y 227.042,Z 592.062,A -85,B 0,C 180,E1 -19895.329,E2 -19895.329} C_VEL
LIN {X 0,Y 226.769,Z 590.26,A -85,B 0,C 180,E1 -19897.368,E2 -19897.368} C_VEL
LIN {X 0,Y 226.705,Z 586.043,A -85,B 0,C 180,E1 -19900.72,E2 -19900.72} C_VEL
LIN {X 0,Y 227.236,Z 581.469,A -85,B 0,C 180,E1 -19903.413,E2 -19903.413} C_VEL
LIN {X 0,Y 228.212,Z 575.701,A -85,B 0,C 180,E1 -19906.091,E2 -19906.091} C_VEL
LIN {X 0,Y 229.535,Z 569.919,A -85,B 0,C 180,E1 -19908.268,E2 -19908.268} C_VEL
LIN {X 0,Y 231.682,Z 561.374,A -85,B 0,C 180,E1 -19910.882,E2 -19910.882} C_VEL
LIN {X 0,Y 233.046,Z 554.493,A -85,B 0,C 180,E1 -19912.613,E2 -19912.613} C_VEL
LIN {X 0,Y 234.189,Z 544.145,A -85,B 0,C 180,E1 -19914.844,E2 -19914.844} C_VEL
LIN {X 0,Y 234.882,Z 532.421,A -85,B 0,C 180,E1 -19916.908,E2 -19916.908} C_VEL
LIN {X 0,Y 234.899,Z 520.902,A -85,B 0,C 180,E1 -19918.601,E2 -19918.601} C_VEL
LIN {X 0,Y 234.336,Z 509.38,A -85,B 0,C 180,E1 -19920.021,E2 -19920.021} C_VEL
LIN {X 0,Y 232.658,Z 496.04,A -85,B 0,C 180,E1 -19921.428,E2 -19921.428} C_VEL
LIN {X 0,Y 230.13,Z 483.023,A -85,B 0,C 180,E1 -19922.566,E2 -19922.566} C_VEL
LIN {X 0,Y 229.902,Z 480.975,A -85,B 0,C 180,E1 -19922.733,E2 -19922.733} C_VEL
LIN {X 0,Y 231.831,Z 472.717,A -85,B 0,C 180,E1 -19927.323,E2 -19927.323} C_VEL
LIN {X 0,Y 232.671,Z 469.088,A -85,B 0,C 180,E1 -19929.37,E2 -19929.37} C_VEL
LIN {X 0,Y 232.543,Z 466.474,A -85,B 0,C 180,E1 -19930.926,E2 -19930.926} C_VEL
LIN {X 0,Y 231.303,Z 460.105,A -85,B 0,C 180,E1 -19934.948,E2 -19934.948} C_VEL
LIN {X 0,Y 230.156,Z 454.157,A -85,B 0,C 180,E1 -19938.966,E2 -19938.966} C_VEL
LIN {X 0,Y 229.108,Z 448.651,A -85,B 0,C 180,E1 -19942.898,E2 -19942.898} C_VEL
LIN {X 0,Y 227.939,Z 443.092,A -85,B 0,C 180,E1 -19947.345,E2 -19947.345} C_VEL
LIN {X 0,Y 227.906,Z 443.101,A -85,B 0,C 180,E1 -19950.436,E2 -19950.436} C_VEL
LIN {X 0,Y 227.927,Z 443.091,A -85,B 0,C 180,E1 -19954.426,E2 -19954.426} C_VEL
LIN {X 0,Y 227.95,Z 443.086,A -85,B 0,C 180,E1 -19958.286,E2 -19958.286} C_VEL
LIN {X 0,Y 228.037,Z 443.08,A -85,B 0,C 180,E1 -19962.826,E2 -19962.826} C_VEL
LIN {X 0,Y 228.076,Z 443.079,A -85,B 0,C 180,E1 -19967.543,E2 -19967.543} C_VEL
LIN {X 0,Y 228.266,Z 443.052,A -85,B 0,C 180,E1 -19971.145,E2 -19971.145} C_VEL
LIN {X 0,Y 228.322,Z 443.046,A -85,B 0,C 180,E1 -19972.928,E2 -19972.928} C_VEL
LIN {X 0,Y 228.559,Z 443.015,A -85,B 0,C 180,E1 -19978.238,E2 -19978.238} C_VEL
LIN {X 0,Y 228.558,Z 443.016,A -85,B 0,C 180,E1 -19981.762,E2 -19981.762} C_VEL
LIN {X 0,Y 228.322,Z 443.042,A -85,B 0,C 180,E1 -19987.073,E2 -19987.073} C_VEL
LIN {X 0,Y 228.149,Z 443.062,A -85,B 0,C 180,E1 -19990.651,E2 -19990.651} C_VEL
LIN {X 0,Y 228.068,Z 443.04,A -85,B 0,C 180,E1 -19994.272,E2 -19994.272} C_VEL
LIN {X 0,Y 228.006,Z 443.056,A -85,B 0,C 180,E1 -19997.953,E2 -19997.953} C_VEL
LIN {X 0,Y 227.933,Z 443.089,A -85,B 0,C 180,E1 -20002.329,E2 -20002.329} C_VEL
LIN {X 0,Y 227.944,Z 443.06,A -85,B 0,C 180,E1 -20006.602,E2 -20006.602} C_VEL
LIN {X 0,Y 227.899,Z 443.083,A -85,B 0,C 180,E1 -20010.291,E2 -20010.291} C_VEL
LIN {X 0,Y 227.879,Z 443.096,A -85,B 0,C 180,E1 -20013.72,E2 -20013.72} C_VEL
LIN {X 0,Y 227.846,Z 443.102,A -85,B 0,C 180,E1 -20018.091,E2 -20018.091} C_VEL
LIN {X 0,Y 227.847,Z 443.103,A -85,B 0,C 180,E1 -20022.734,E2 -20022.734} C_VEL
LIN {X 0,Y 227.92,Z 443.089,A -85,B 0,C 180,E1 -20027.736,E2 -20027.736} C_VEL
LIN {X 0,Y 227.883,Z 443.094,A -85,B 0,C 180,E1 -20031.916,E2 -20031.916} C_VEL
LIN {X 0,Y 227.893,Z 443.09,A -85,B 0,C 180,E1 -20036.373,E2 -20036.373} C_VEL
LIN {X 0,Y 227.933,Z 443.168,A -85,B 0,C 180,E1 -20038.16,E2 -20038.16} C_VEL
LIN {X 0,Y 228.743,Z 445.601,A -85,B 0,C 180,E1 -20038.512,E2 -20038.512} C_VEL
LIN {X 0,Y 233.14,Z 454.767,A -85,B 0,C 180,E1 -20040.224,E2 -20040.224} C_VEL
LIN {X 0,Y 236.756,Z 463.936,A -85,B 0,C 180,E1 -20042.02,E2 -20042.02} C_VEL
LIN {X 0,Y 239.504,Z 472.862,A -85,B 0,C 180,E1 -20043.886,E2 -20043.886} C_VEL
LIN {X 0,Y 241.371,Z 480.378,A -85,B 0,C 180,E1 -20045.606,E2 -20045.606} C_VEL
LIN {X 0,Y 240.606,Z 485.184,A -85,B 0,C 180,E1 -20046.548,E2 -20046.548} C_VEL
LIN {X 0,Y 238.665,Z 493.595,A -85,B 0,C 180,E1 -20048.402,E2 -20048.402} C_VEL
LIN {X 0,Y 236.651,Z 501.338,A -85,B 0,C 180,E1 -20050.482,E2 -20050.482} C_VEL
LIN {X 0,Y 234.463,Z 508.904,A -85,B 0,C 180,E1 -20053.007,E2 -20053.007} C_VEL
LIN {X 0,Y 233.032,Z 514.062,A -85,B 0,C 180,E1 -20055.159,E2 -20055.159} C_VEL
LIN {X 0,Y 231.609,Z 519.006,A -85,B 0,C 180,E1 -20057.736,E2 -20057.736} C_VEL
LIN {X 0,Y 230.301,Z 522.884,A -85,B 0,C 180,E1 -20060.337,E2 -20060.337} C_VEL
LIN {X 0,Y 229.276,Z 525.751,A -85,B 0,C 180,E1 -20062.957,E2 -20062.957} C_VEL
LIN {X 0,Y 228.789,Z 527.121,A -85,B 0,C 180,E1 -20064.712,E2 -20064.712} C_VEL
LIN {X 0,Y 228.574,Z 528.643,A -85,B 0,C 180,E1 -20068.238,E2 -20068.238} C_VEL
LIN {X 0,Y 228.537,Z 528.864,A -85,B 0,C 180,E1 -20070,E2 -20070} C_VEL
LIN {X 0,Y 228.573,Z 528.678,A -85,B 0,C 180,E1 -20071.762,E2 -20071.762} C_VEL
LIN {X 0,Y 228.779,Z 527.2,A -85,B 0,C 180,E1 -20075.288,E2 -20075.288} C_VEL
LIN {X 0,Y 229.261,Z 525.866,A -85,B 0,C 180,E1 -20077.043,E2 -20077.043} C_VEL
LIN {X 0,Y 230.289,Z 523.042,A -85,B 0,C 180,E1 -20079.663,E2 -20079.663} C_VEL
LIN {X 0,Y 231.57,Z 519.221,A -85,B 0,C 180,E1 -20082.266,E2 -20082.266} C_VEL
LIN {X 0,Y 233.186,Z 513.301,A -85,B 0,C 180,E1 -20085.322,E2 -20085.322} C_VEL
LIN {X 0,Y 235.141,Z 506.904,A -85,B 0,C 180,E1 -20087.84,E2 -20087.84} C_VEL
LIN {X 0,Y 237.408,Z 498.863,A -85,B 0,C 180,E1 -20090.355,E2 -20090.355} C_VEL
LIN {X 0,Y 239.375,Z 490.634,A -85,B 0,C 180,E1 -20092.438,E2 -20092.438} C_VEL
LIN {X 0,Y 241.491,Z 481.32,A -85,B 0,C 180,E1 -20094.323,E2 -20094.323} C_VEL
LIN {X 0,Y 239.784,Z 473.611,A -85,B 0,C 180,E1 -20096.081,E2 -20096.081} C_VEL
LIN {X 0,Y 236.899,Z 464.322,A -85,B 0,C 180,E1 -20098.044,E2 -20098.044} C_VEL
LIN {X 0,Y 233.539,Z 455.577,A -85,B 0,C 180,E1 -20099.759,E2 -20099.759} C_VEL
LIN {X 0,Y 229.073,Z 446.189,A -85,B 0,C 180,E1 -20101.522,E2 -20101.522} C_VEL
LIN {X 0,Y 227.962,Z 443.462,A -85,B 0,C 180,E1 -20101.959,E2 -20101.959} C_VEL
LIN {X 0,Y 227.924,Z 443.087,A -85,B 0,C 180,E1 -20102.044,E2 -20102.044} C_VEL
LIN {X 0,Y 227.913,Z 443.096,A -85,B 0,C 180,E1 -20106.703,E2 -20106.703} C_VEL
LIN {X 0,Y 227.917,Z 443.094,A -85,B 0,C 180,E1 -20110.357,E2 -20110.357} C_VEL
LIN {X 0,Y 227.925,Z 443.094,A -85,B 0,C 180,E1 -20112.716,E2 -20112.716} C_VEL
LIN {X 0,Y 227.833,Z 443.104,A -85,B 0,C 180,E1 -20117.76,E2 -20117.76} C_VEL
LIN {X 0,Y 227.848,Z 443.102,A -85,B 0,C 180,E1 -20121.909,E2 -20121.909} C_VEL
LIN {X 0,Y 227.88,Z 443.1,A -85,B 0,C 180,E1 -20126.377,E2 -20126.377} C_VEL
LIN {X 0,Y 227.906,Z 443.097,A -85,B 0,C 180,E1 -20130.436,E2 -20130.436} C_VEL
LIN {X 0,Y 227.93,Z 443.092,A -85,B 0,C 180,E1 -20134.426,E2 -20134.426} C_VEL
LIN {X 0,Y 227.964,Z 443.083,A -85,B 0,C 180,E1 -20138.287,E2 -20138.287} C_VEL
LIN {X 0,Y 228.037,Z 443.074,A -85,B 0,C 180,E1 -20142.825,E2 -20142.825} C_VEL
LIN {X 0,Y 228.075,Z 443.069,A -85,B 0,C 180,E1 -20147.543,E2 -20147.543} C_VEL
LIN {X 0,Y 228.265,Z 443.05,A -85,B 0,C 180,E1 -20151.144,E2 -20151.144} C_VEL
LIN {X 0,Y 228.321,Z 443.038,A -85,B 0,C 180,E1 -20152.927,E2 -20152.927} C_VEL
LIN {X 0,Y 228.557,Z 443.015,A -85,B 0,C 180,E1 -20158.238,E2 -20158.238} C_VEL
LIN {X 0,Y 228.557,Z 443.004,A -85,B 0,C 180,E1 -20161.762,E2 -20161.762} C_VEL
LIN {X 0,Y 228.321,Z 443.037,A -85,B 0,C 180,E1 -20167.072,E2 -20167.072} C_VEL
LIN {X 0,Y 228.147,Z 443.065,A -85,B 0,C 180,E1 -20170.651,E2 -20170.651} C_VEL
LIN {X 0,Y 228.067,Z 443.075,A -85,B 0,C 180,E1 -20174.272,E2 -20174.272} C_VEL
LIN {X 0,Y 228.005,Z 443.081,A -85,B 0,C 180,E1 -20177.953,E2 -20177.953} C_VEL
LIN {X 0,Y 227.918,Z 443.097,A -85,B 0,C 180,E1 -20182.321,E2 -20182.321} C_VEL
LIN {X 0,Y 227.943,Z 443.093,A -85,B 0,C 180,E1 -20186.602,E2 -20186.602} C_VEL
LIN {X 0,Y 227.898,Z 443.096,A -85,B 0,C 180,E1 -20190.291,E2 -20190.291} C_VEL
LIN {X 0,Y 227.935,Z 443.134,A -85,B 0,C 180,E1 -20192.655,E2 -20192.655} C_VEL
LIN {X 0,Y 229.132,Z 448.828,A -85,B 0,C 180,E1 -20197.11,E2 -20197.11} C_VEL
LIN {X 0,Y 230.162,Z 454.253,A -85,B 0,C 180,E1 -20201.033,E2 -20201.033} C_VEL
LIN {X 0,Y 231.532,Z 461.251,A -85,B 0,C 180,E1 -20205.721,E2 -20205.721} C_VEL
LIN {X 0,Y 232.547,Z 466.555,A -85,B 0,C 180,E1 -20209.073,E2 -20209.073} C_VEL
LIN {X 0,Y 232.67,Z 469.171,A -85,B 0,C 180,E1 -20210.63,E2 -20210.63} C_VEL
LIN {X 0,Y 231.003,Z 476.433,A -85,B 0,C 180,E1 -20214.686,E2 -20214.686} C_VEL
LIN {X 0,Y 229.923,Z 481.053,A -85,B 0,C 180,E1 -20217.255,E2 -20217.255} C_VEL
LIN {X 0,Y 232.711,Z 495.865,A -85,B 0,C 180,E1 -20218.516,E2 -20218.516} C_VEL
LIN {X 0,Y 232.982,Z 497.697,A -85,B 0,C 180,E1 -20218.696,E2 -20218.696} C_VEL
LIN {X 0,Y 232.988,Z 503.485,A -85,B 0,C 180,E1 -20219.183,E2 -20219.183} C_VEL
LIN {X 0,Y 231.079,Z 512.995,A -85,B 0,C 180,E1 -20219.915,E2 -20219.915} C_VEL
LIN {X 0,Y 228.934,Z 521.82,A -85,B 0,C 180,E1 -20220.794,E2 -20220.794} C_VEL
LIN {X 0,Y 228.421,Z 526.853,A -85,B 0,C 180,E1 -20221.483,E2 -20221.483} C_VEL
LIN {X 0,Y 227.922,Z 538.294,A -85,B 0,C 180,E1 -20223.409,E2 -20223.409} C_VEL
LIN {X 0,Y 226.94,Z 548.724,A -85,B 0,C 180,E1 -20225.531,E2 -20225.531} C_VEL
LIN {X 0,Y 225.748,Z 557.192,A -85,B 0,C 180,E1 -20227.582,E2 -20227.582} C_VEL
LIN {X 0,Y 223.604,Z 565.95,A -85,B 0,C 180,E1 -20230.12,E2 -20230.12} C_VEL
LIN {X 0,Y 221.57,Z 573.706,A -85,B 0,C 180,E1 -20232.938,E2 -20232.938} C_VEL
LIN {X 0,Y 220.286,Z 580.52,A -85,B 0,C 180,E1 -20236.156,E2 -20236.156} C_VEL
LIN {X 0,Y 219.691,Z 585.077,A -85,B 0,C 180,E1 -20238.934,E2 -20238.934} C_VEL
LIN {X 0,Y 219.72,Z 589.445,A -85,B 0,C 180,E1 -20242.556,E2 -20242.556} C_VEL
LIN {X 0,Y 219.962,Z 591.066,A -85,B 0,C 180,E1 -20244.5,E2 -20244.5} C_VEL
LIN {X 0,Y 220.282,Z 592.18,A -85,B 0,C 180,E1 -20246.342,E2 -20246.342} C_VEL
LIN {X 0,Y 221.038,Z 593.163,A -85,B 0,C 180,E1 -20250,E2 -20250} C_VEL
LIN {X 0,Y 220.282,Z 592.164,A -85,B 0,C 180,E1 -20253.659,E2 -20253.659} C_VEL
LIN {X 0,Y 219.942,Z 591.042,A -85,B 0,C 180,E1 -20255.501,E2 -20255.501} C_VEL
LIN {X 0,Y 219.698,Z 589.453,A -85,B 0,C 180,E1 -20257.398,E2 -20257.398} C_VEL
LIN {X 0,Y 219.619,Z 586.329,A -85,B 0,C 180,E1 -20260.137,E2 -20260.137} C_VEL
LIN {X 0,Y 219.992,Z 582.113,A -85,B 0,C 180,E1 -20262.922,E2 -20262.922} C_VEL
LIN {X 0,Y 221.095,Z 575.719,A -85,B 0,C 180,E1 -20266.149,E2 -20266.149} C_VEL
LIN {X 0,Y 222.414,Z 570.093,A -85,B 0,C 180,E1 -20268.421,E2 -20268.421} C_VEL
LIN {X 0,Y 224.591,Z 561.867,A -85,B 0,C 180,E1 -20271.092,E2 -20271.092} C_VEL
LIN {X 0,Y 226.038,Z 555.29,A -85,B 0,C 180,E1 -20272.871,E2 -20272.871} C_VEL
LIN {X 0,Y 227.284,Z 545.31,A -85,B 0,C 180,E1 -20275.162,E2 -20275.162} C_VEL
LIN {X 0,Y 228.11,Z 534.607,A -85,B 0,C 180,E1 -20277.205,E2 -20277.205} C_VEL
LIN {X 0,Y 228.364,Z 523.451,A -85,B 0,C 180,E1 -20278.994,E2 -20278.994} C_VEL
LIN {X 0,Y 228.01,Z 512.254,A -85,B 0,C 180,E1 -20280.509,E2 -20280.509} C_VEL
LIN {X 0,Y 226.673,Z 499.345,A -85,B 0,C 180,E1 -20281.999,E2 -20281.999} C_VEL
LIN {X 0,Y 224.35,Z 485.828,A -85,B 0,C 180,E1 -20283.315,E2 -20283.315} C_VEL
LIN {X 0,Y 223.21,Z 479.922,A -85,B 0,C 180,E1 -20283.814,E2 -20283.814} C_VEL
LIN {X 0,Y 225.378,Z 471.318,A -85,B 0,C 180,E1 -20288.778,E2 -20288.778} C_VEL
LIN {X 0,Y 225.691,Z 469.771,A -85,B 0,C 180,E1 -20289.681,E2 -20289.681} C_VEL
LIN {X 0,Y 225.39,Z 466.785,A -85,B 0,C 180,E1 -20291.552,E2 -20291.552} C_VEL
LIN {X 0,Y 224.297,Z 461.267,A -85,B 0,C 180,E1 -20295.172,E2 -20295.172} C_VEL
LIN {X 0,Y 222.997,Z 454.442,A -85,B 0,C 180,E1 -20299.981,E2 -20299.981} C_VEL
LIN {X 0,Y 221.946,Z 448.917,A -85,B 0,C 180,E1 -20304.14,E2 -20304.14} C_VEL
LIN {X 0,Y 220.829,Z 443.978,A -85,B 0,C 180,E1 -20308.325,E2 -20308.325} C_VEL
LIN {X 0,Y 220.896,Z 443.972,A -85,B 0,C 180,E1 -20313.55,E2 -20313.55} C_VEL
LIN {X 0,Y 220.868,Z 443.968,A -85,B 0,C 180,E1 -20317.552,E2 -20317.552} C_VEL
LIN {X 0,Y 220.987,Z 443.959,A -85,B 0,C 180,E1 -20322.571,E2 -20322.571} C_VEL
LIN {X 0,Y 221.015,Z 443.958,A -85,B 0,C 180,E1 -20327.139,E2 -20327.139} C_VEL
LIN {X 0,Y 221.204,Z 443.931,A -85,B 0,C 180,E1 -20330.859,E2 -20330.859} C_VEL
LIN {X 0,Y 221.142,Z 443.939,A -85,B 0,C 180,E1 -20334.529,E2 -20334.529} C_VEL
LIN {X 0,Y 221.517,Z 443.893,A -85,B 0,C 180,E1 -20338.182,E2 -20338.182} C_VEL
LIN {X 0,Y 221.516,Z 443.893,A -85,B 0,C 180,E1 -20341.818,E2 -20341.818} C_VEL
LIN {X 0,Y 221.257,Z 443.922,A -85,B 0,C 180,E1 -20347.3,E2 -20347.3} C_VEL
LIN {X 0,Y 221.085,Z 443.94,A -85,B 0,C 180,E1 -20350.996,E2 -20350.996} C_VEL
LIN {X 0,Y 221.019,Z 443.911,A -85,B 0,C 180,E1 -20356.63,E2 -20356.63} C_VEL
LIN {X 0,Y 220.896,Z 443.962,A -85,B 0,C 180,E1 -20360.486,E2 -20360.486} C_VEL
LIN {X 0,Y 220.87,Z 443.962,A -85,B 0,C 180,E1 -20364.435,E2 -20364.435} C_VEL
LIN {X 0,Y 220.829,Z 443.941,A -85,B 0,C 180,E1 -20368.515,E2 -20368.515} C_VEL
LIN {X 0,Y 220.819,Z 443.977,A -85,B 0,C 180,E1 -20372.756,E2 -20372.756} C_VEL
LIN {X 0,Y 220.812,Z 443.98,A -85,B 0,C 180,E1 -20377.278,E2 -20377.278} C_VEL
